// ---- Nodes/Algebraic Image Ops/Node_F_VN_BitwiseXorImagesExp.TcPOU
{attribute 'linkalways'} 
{attribute 'no_explicit_call' := 'This FB is a CLASS and must be accessed using methods or properties'}
{attribute 'enable_dynamic_creation'}
FUNCTION_BLOCK Node_F_VN_BitwiseXorImagesExp EXTENDS VisionNode
VAR
    ipSrcImage1 : _ITcVnImage;
    ipSrcImage2 : _ITcVnImage;
    ipDestImage : _ITcVnImage;
    ipMask : _ITcVnImage;
    hrPrev : _HRESULT(S_OK);
	hresult : _HRESULT(S_OK);
END_VAR

METHOD PUBLIC  Clone : I_Node
VAR
	pNode : POINTER TO Node_F_VN_BitwiseXorImagesExp;
END_VAR
pNode := __NEW(Node_F_VN_BitwiseXorImagesExp);
Clone := pNode^;
END_METHOD

METHOD FB_init : BOOL
VAR_INPUT
	bInitRetains : BOOL; // if TRUE, the retain variables are initialized (warm start / cold start)
	bInCopyCode : BOOL;  // if TRUE, the instance afterwards gets moved into the copy code (online change)
END_VAR
AddInput('ipSrcImage1', ipSrcImage1);
AddInput('ipSrcImage2', ipSrcImage2);
AddInput('ipMask', ipMask);
AddInput('hrPrev', hrPrev);
AddOutput('ipDestImage', ipDestImage);
AddOutput('hresult',hresult);
END_METHOD

METHOD PROTECTED OnExecute
hresult.Value := F_VN_BitwiseXorImagesExp(
    ipSrcImage1 := ipSrcImage1.Value,
    ipSrcImage2 := ipSrcImage2.Value,
	ipDestImage := ipDestImage.Value,
    ipMask := ipMask.Value,
	hrPrev:= hrPrev.Value);
END_METHOD

METHOD PUBLIC PreExecutionCheck
VAR_INPUT
	Check : I_PreExecutionChecks;
END_VAR
Check.IsTrue(ipSrcImage1.IsValid, 'ipSrcImage1 must contain an image');
Check.IsTrue(ipSrcImage2.IsValid, 'ipSrcImage2 must contain an image');
Check.IsTrue(IsImage1SizeEqualToImage2Size(ipSrcImage1.Value, ipSrcImage2.Value), 'ipSrcImage1 must be the same size as ipSrcImage2');
Check.IsTrue(ipMask.IsValid, 'ipMask must contain an image');
Check.IsTrue(ipMask.HasChannelCount(1), 'ipMask must have 1 channel');
Check.IsTrue(ipMask.IsPixelDepth(8), 'ipMask must have 8 bit pixel depth');
Check.IsTrue(IsImage1SizeEqualToImage2Size(ipMask.Value, ipSrcImage1.Value), 'ipMask must be the same size as ipSrcImage1');
END_METHOD

END_FUNCTION_BLOCK

// ---- Nodes/Algebraic Image Ops/Node_F_VN_BitwiseOrImagesExp.TcPOU
{attribute 'linkalways'} 
{attribute 'no_explicit_call' := 'This FB is a CLASS and must be accessed using methods or properties'}
{attribute 'enable_dynamic_creation'}
FUNCTION_BLOCK Node_F_VN_BitwiseOrImagesExp EXTENDS VisionNode
VAR
    ipSrcImage1 : _ITcVnImage;
    ipSrcImage2 : _ITcVnImage;
    ipDestImage : _ITcVnImage;
    ipMask : _ITcVnImage;
    hrPrev : _HRESULT(S_OK);
	hresult : _HRESULT(S_OK);
END_VAR

METHOD PUBLIC  Clone : I_Node
VAR
	pNode : POINTER TO Node_F_VN_BitwiseOrImagesExp;
END_VAR
pNode := __NEW(Node_F_VN_BitwiseOrImagesExp);
Clone := pNode^;
END_METHOD

METHOD FB_init : BOOL
VAR_INPUT
	bInitRetains : BOOL; // if TRUE, the retain variables are initialized (warm start / cold start)
	bInCopyCode : BOOL;  // if TRUE, the instance afterwards gets moved into the copy code (online change)
END_VAR
AddInput('ipSrcImage1', ipSrcImage1);
AddInput('ipSrcImage2', ipSrcImage2);
AddInput('ipMask', ipMask);
AddInput('hrPrev', hrPrev);
AddOutput('ipDestImage', ipDestImage);
AddOutput('hresult',hresult);
END_METHOD

METHOD PROTECTED OnExecute
hresult.Value := F_VN_BitwiseOrImagesExp(
    ipSrcImage1 := ipSrcImage1.Value,
    ipSrcImage2 := ipSrcImage2.Value,
	ipDestImage := ipDestImage.Value,
    ipMask := ipMask.Value,
	hrPrev:= hrPrev.Value);
END_METHOD

METHOD PUBLIC PreExecutionCheck
VAR_INPUT
	Check : I_PreExecutionChecks;
END_VAR
Check.IsTrue(ipSrcImage1.IsValid, 'ipSrcImage1 must contain an image');
Check.IsTrue(ipSrcImage2.IsValid, 'ipSrcImage2 must contain an image');
Check.IsTrue(IsImage1SizeEqualToImage2Size(ipSrcImage1.Value, ipSrcImage2.Value), 'ipSrcImage1 must be the same size as ipSrcImage2');
Check.IsTrue(ipMask.IsValid, 'ipMask must contain an image');
Check.IsTrue(ipMask.HasChannelCount(1), 'ipMask must have 1 channel');
Check.IsTrue(ipMask.IsPixelDepth(8), 'ipMask must have 8 bit pixel depth');
Check.IsTrue(IsImage1SizeEqualToImage2Size(ipMask.Value, ipSrcImage1.Value), 'ipMask must be the same size as ipSrcImage1');
END_METHOD

END_FUNCTION_BLOCK

// ---- Nodes/Algebraic Image Ops/Node_F_VN_BitwiseAndScalarWithImage.TcPOU
{attribute 'linkalways'} 
{attribute 'no_explicit_call' := 'This FB is a CLASS and must be accessed using methods or properties'}
{attribute 'enable_dynamic_creation'}
FUNCTION_BLOCK Node_F_VN_BitwiseAndScalarWithImage EXTENDS VisionNode
VAR
    fScalar : _LREAL(0.0);
    ipSrcImage : _ITcVnImage;
    ipDestImage : _ITcVnImage;
    hrPrev : _HRESULT(S_OK);
	hresult : _HRESULT(S_OK);
END_VAR

METHOD PUBLIC  Clone : I_Node
VAR
	pNode : POINTER TO Node_F_VN_BitwiseAndScalarWithImage;
END_VAR
pNode := __NEW(Node_F_VN_BitwiseAndScalarWithImage);
Clone := pNode^;
END_METHOD

METHOD FB_init : BOOL
VAR_INPUT
	bInitRetains : BOOL; // if TRUE, the retain variables are initialized (warm start / cold start)
	bInCopyCode : BOOL;  // if TRUE, the instance afterwards gets moved into the copy code (online change)
END_VAR
AddParameter('fScalar', fScalar);
AddInput('ipSrcImage', ipSrcImage);
AddInput('hrPrev', hrPrev);
AddOutput('ipDestImage', ipDestImage);
AddOutput('hresult',hresult);
END_METHOD

METHOD PROTECTED OnExecute
hresult.Value := F_VN_BitwiseAndScalarWithImage(
    fScalar := fScalar.Value,
    ipSrcImage := ipSrcImage.Value,
	ipDestImage := ipDestImage.Value,
	hrPrev:= hrPrev.Value);
END_METHOD

METHOD PUBLIC PreExecutionCheck
VAR_INPUT
	Check : I_PreExecutionChecks;
END_VAR
Check.IsTrue(ipSrcImage.IsValid, 'ipSrcImage must contain an image');
END_METHOD

END_FUNCTION_BLOCK

// ---- Nodes/Algebraic Image Ops/Node_F_VN_BitwiseXorVectorWithImage.TcPOU
{attribute 'linkalways'} 
{attribute 'no_explicit_call' := 'This FB is a CLASS and must be accessed using methods or properties'}
{attribute 'enable_dynamic_creation'}
FUNCTION_BLOCK Node_F_VN_BitwiseXorVectorWithImage EXTENDS VisionNode
VAR
    aVector : _TcVnVector4_LREAL;
    ipSrcImage : _ITcVnImage;
    ipDestImage : _ITcVnImage;
    hrPrev : _HRESULT(S_OK);
	hresult : _HRESULT(S_OK);
END_VAR

METHOD PUBLIC  Clone : I_Node
VAR
	pNode : POINTER TO Node_F_VN_BitwiseXorVectorWithImage;
END_VAR
pNode := __NEW(Node_F_VN_BitwiseXorVectorWithImage);
Clone := pNode^;
END_METHOD

METHOD FB_init : BOOL
VAR_INPUT
	bInitRetains : BOOL; // if TRUE, the retain variables are initialized (warm start / cold start)
	bInCopyCode : BOOL;  // if TRUE, the instance afterwards gets moved into the copy code (online change)
END_VAR
AddInput('aVector', aVector);
AddInput('ipSrcImage', ipSrcImage);
AddInput('hrPrev', hrPrev);
AddOutput('ipDestImage', ipDestImage);
AddOutput('hresult',hresult);
END_METHOD

METHOD PROTECTED OnExecute
hresult.Value := F_VN_BitwiseXorVectorWithImage(
    aVector := aVector.Value,
    ipSrcImage := ipSrcImage.Value,
	ipDestImage := ipDestImage.Value,
	hrPrev:= hrPrev.Value);
END_METHOD

METHOD PUBLIC PreExecutionCheck
VAR_INPUT
	Check : I_PreExecutionChecks;
END_VAR
Check.IsTrue(ipSrcImage.IsValid, 'ipSrcImage must contain an image');
END_METHOD

END_FUNCTION_BLOCK

// ---- Nodes/Algebraic Image Ops/Node_F_VN_BitwiseXorScalarWithImage.TcPOU
{attribute 'linkalways'} 
{attribute 'no_explicit_call' := 'This FB is a CLASS and must be accessed using methods or properties'}
{attribute 'enable_dynamic_creation'}
FUNCTION_BLOCK Node_F_VN_BitwiseXorScalarWithImage EXTENDS VisionNode
VAR
    fScalar : _LREAL(0.0);
    ipSrcImage : _ITcVnImage;
    ipDestImage : _ITcVnImage;
    hrPrev : _HRESULT(S_OK);
	hresult : _HRESULT(S_OK);
END_VAR

METHOD PUBLIC  Clone : I_Node
VAR
	pNode : POINTER TO Node_F_VN_BitwiseXorScalarWithImage;
END_VAR
pNode := __NEW(Node_F_VN_BitwiseXorScalarWithImage);
Clone := pNode^;
END_METHOD

METHOD FB_init : BOOL
VAR_INPUT
	bInitRetains : BOOL; // if TRUE, the retain variables are initialized (warm start / cold start)
	bInCopyCode : BOOL;  // if TRUE, the instance afterwards gets moved into the copy code (online change)
END_VAR
AddParameter('fScalar', fScalar);
AddInput('ipSrcImage', ipSrcImage);
AddInput('hrPrev', hrPrev);
AddOutput('ipDestImage', ipDestImage);
AddOutput('hresult',hresult);
END_METHOD

METHOD PROTECTED OnExecute
hresult.Value := F_VN_BitwiseXorScalarWithImage(
    fScalar := fScalar.Value,
    ipSrcImage := ipSrcImage.Value,
	ipDestImage := ipDestImage.Value,
	hrPrev:= hrPrev.Value);
END_METHOD

METHOD PUBLIC PreExecutionCheck
VAR_INPUT
	Check : I_PreExecutionChecks;
END_VAR
Check.IsTrue(ipSrcImage.IsValid, 'ipSrcImage must contain an image');
END_METHOD

END_FUNCTION_BLOCK

// ---- Nodes/Algebraic Image Ops/Node_F_VN_BitwiseOrVectorWithImage.TcPOU
{attribute 'linkalways'} 
{attribute 'no_explicit_call' := 'This FB is a CLASS and must be accessed using methods or properties'}
{attribute 'enable_dynamic_creation'}
FUNCTION_BLOCK Node_F_VN_BitwiseOrVectorWithImage EXTENDS VisionNode
VAR
    aVector : _TcVnVector4_LREAL;
    ipSrcImage : _ITcVnImage;
    ipDestImage : _ITcVnImage;
    hrPrev : _HRESULT(S_OK);
	hresult : _HRESULT(S_OK);
END_VAR

METHOD PUBLIC  Clone : I_Node
VAR
	pNode : POINTER TO Node_F_VN_BitwiseOrVectorWithImage;
END_VAR
pNode := __NEW(Node_F_VN_BitwiseOrVectorWithImage);
Clone := pNode^;
END_METHOD

METHOD FB_init : BOOL
VAR_INPUT
	bInitRetains : BOOL; // if TRUE, the retain variables are initialized (warm start / cold start)
	bInCopyCode : BOOL;  // if TRUE, the instance afterwards gets moved into the copy code (online change)
END_VAR
AddInput('aVector', aVector);
AddInput('ipSrcImage', ipSrcImage);
AddInput('hrPrev', hrPrev);
AddOutput('ipDestImage', ipDestImage);
AddOutput('hresult',hresult);
END_METHOD

METHOD PROTECTED OnExecute
hresult.Value := F_VN_BitwiseOrVectorWithImage(
    aVector := aVector.Value,
    ipSrcImage := ipSrcImage.Value,
	ipDestImage := ipDestImage.Value,
	hrPrev:= hrPrev.Value);
END_METHOD

METHOD PUBLIC PreExecutionCheck
VAR_INPUT
	Check : I_PreExecutionChecks;
END_VAR
Check.IsTrue(ipSrcImage.IsValid, 'ipSrcImage must contain an image');
END_METHOD

END_FUNCTION_BLOCK

// ---- Nodes/Algebraic Image Ops/Node_F_VN_BitwiseOrScalarWithImage.TcPOU
{attribute 'linkalways'} 
{attribute 'no_explicit_call' := 'This FB is a CLASS and must be accessed using methods or properties'}
{attribute 'enable_dynamic_creation'}
FUNCTION_BLOCK Node_F_VN_BitwiseOrScalarWithImage EXTENDS VisionNode
VAR
    fScalar : _LREAL(0.0);
    ipSrcImage : _ITcVnImage;
    ipDestImage : _ITcVnImage;
    hrPrev : _HRESULT(S_OK);
	hresult : _HRESULT(S_OK);
END_VAR

METHOD PUBLIC  Clone : I_Node
VAR
	pNode : POINTER TO Node_F_VN_BitwiseOrScalarWithImage;
END_VAR
pNode := __NEW(Node_F_VN_BitwiseOrScalarWithImage);
Clone := pNode^;
END_METHOD

METHOD FB_init : BOOL
VAR_INPUT
	bInitRetains : BOOL; // if TRUE, the retain variables are initialized (warm start / cold start)
	bInCopyCode : BOOL;  // if TRUE, the instance afterwards gets moved into the copy code (online change)
END_VAR
AddParameter('fScalar', fScalar);
AddInput('ipSrcImage', ipSrcImage);
AddInput('hrPrev', hrPrev);
AddOutput('ipDestImage', ipDestImage);
AddOutput('hresult',hresult);
END_METHOD

METHOD PROTECTED OnExecute
hresult.Value := F_VN_BitwiseOrScalarWithImage(
    fScalar := fScalar.Value,
    ipSrcImage := ipSrcImage.Value,
	ipDestImage := ipDestImage.Value,
	hrPrev:= hrPrev.Value);
END_METHOD

METHOD PUBLIC PreExecutionCheck
VAR_INPUT
	Check : I_PreExecutionChecks;
END_VAR
Check.IsTrue(ipSrcImage.IsValid, 'ipSrcImage must contain an image');
END_METHOD

END_FUNCTION_BLOCK

// ---- Nodes/Algebraic Image Ops/Node_F_VN_BitwiseAndVectorWithImage.TcPOU
{attribute 'linkalways'} 
{attribute 'no_explicit_call' := 'This FB is a CLASS and must be accessed using methods or properties'}
{attribute 'enable_dynamic_creation'}
FUNCTION_BLOCK Node_F_VN_BitwiseAndVectorWithImage EXTENDS VisionNode
VAR
    aVector : _TcVnVector4_LREAL;
    ipSrcImage : _ITcVnImage;
    ipDestImage : _ITcVnImage;
    hrPrev : _HRESULT(S_OK);
	hresult : _HRESULT(S_OK);
END_VAR

METHOD PUBLIC  Clone : I_Node
VAR
	pNode : POINTER TO Node_F_VN_BitwiseAndVectorWithImage;
END_VAR
pNode := __NEW(Node_F_VN_BitwiseAndVectorWithImage);
Clone := pNode^;
END_METHOD

METHOD FB_init : BOOL
VAR_INPUT
	bInitRetains : BOOL; // if TRUE, the retain variables are initialized (warm start / cold start)
	bInCopyCode : BOOL;  // if TRUE, the instance afterwards gets moved into the copy code (online change)
END_VAR
AddInput('aVector', aVector);
AddInput('ipSrcImage', ipSrcImage);
AddInput('hrPrev', hrPrev);
AddOutput('ipDestImage', ipDestImage);
AddOutput('hresult',hresult);
END_METHOD

METHOD PROTECTED OnExecute
hresult.Value := F_VN_BitwiseAndVectorWithImage(
    aVector := aVector.Value,
    ipSrcImage := ipSrcImage.Value,
	ipDestImage := ipDestImage.Value,
	hrPrev:= hrPrev.Value);
END_METHOD

METHOD PUBLIC PreExecutionCheck
VAR_INPUT
	Check : I_PreExecutionChecks;
END_VAR
Check.IsTrue(ipSrcImage.IsValid, 'ipSrcImage must contain an image');
END_METHOD

END_FUNCTION_BLOCK

// ---- Nodes/Algebraic Image Ops/Node_F_VN_DivideImageByScalar.TcPOU
{attribute 'linkalways'} 
{attribute 'no_explicit_call' := 'This FB is a CLASS and must be accessed using methods or properties'}
{attribute 'enable_dynamic_creation'}
FUNCTION_BLOCK Node_F_VN_DivideImageByScalar EXTENDS VisionNode
VAR
    ipSrcImage : _ITcVnImage;
    fScalar : _LREAL(0.0);
    ipDestImage : _ITcVnImage;
    hrPrev : _HRESULT(S_OK);
	hresult : _HRESULT(S_OK);
END_VAR

METHOD PUBLIC  Clone : I_Node
VAR
	pNode : POINTER TO Node_F_VN_DivideImageByScalar;
END_VAR
pNode := __NEW(Node_F_VN_DivideImageByScalar);
Clone := pNode^;
END_METHOD

METHOD FB_init : BOOL
VAR_INPUT
	bInitRetains : BOOL; // if TRUE, the retain variables are initialized (warm start / cold start)
	bInCopyCode : BOOL;  // if TRUE, the instance afterwards gets moved into the copy code (online change)
END_VAR
AddInput('ipSrcImage', ipSrcImage);
AddParameter('fScalar', fScalar);
AddInput('hrPrev', hrPrev);
AddOutput('ipDestImage', ipDestImage);
AddOutput('hresult',hresult);
END_METHOD

METHOD PROTECTED OnExecute
hresult.Value := F_VN_DivideImageByScalar(
    ipSrcImage := ipSrcImage.Value,
    fScalar := fScalar.Value,
	ipDestImage := ipDestImage.Value,
	hrPrev:= hrPrev.Value);
END_METHOD

METHOD PUBLIC PreExecutionCheck
VAR_INPUT
	Check : I_PreExecutionChecks;
END_VAR
Check.IsTrue(ipSrcImage.IsValid, 'ipSrcImage must contain an image');
END_METHOD

END_FUNCTION_BLOCK

// ---- Nodes/Algebraic Image Ops/Node_F_VN_DivideVectorByImage.TcPOU
{attribute 'linkalways'} 
{attribute 'no_explicit_call' := 'This FB is a CLASS and must be accessed using methods or properties'}
{attribute 'enable_dynamic_creation'}
FUNCTION_BLOCK Node_F_VN_DivideVectorByImage EXTENDS VisionNode
VAR
    aVector : _TcVnVector4_LREAL;
    ipSrcImage : _ITcVnImage;
    ipDestImage : _ITcVnImage;
    hrPrev : _HRESULT(S_OK);
	hresult : _HRESULT(S_OK);
END_VAR

METHOD PUBLIC  Clone : I_Node
VAR
	pNode : POINTER TO Node_F_VN_DivideVectorByImage;
END_VAR
pNode := __NEW(Node_F_VN_DivideVectorByImage);
Clone := pNode^;
END_METHOD

METHOD FB_init : BOOL
VAR_INPUT
	bInitRetains : BOOL; // if TRUE, the retain variables are initialized (warm start / cold start)
	bInCopyCode : BOOL;  // if TRUE, the instance afterwards gets moved into the copy code (online change)
END_VAR
AddInput('aVector', aVector);
AddInput('ipSrcImage', ipSrcImage);
AddInput('hrPrev', hrPrev);
AddOutput('ipDestImage', ipDestImage);
AddOutput('hresult',hresult);
END_METHOD

METHOD PROTECTED OnExecute
hresult.Value := F_VN_DivideVectorByImage(
    aVector := aVector.Value,
    ipSrcImage := ipSrcImage.Value,
	ipDestImage := ipDestImage.Value,
	hrPrev:= hrPrev.Value);
END_METHOD

METHOD PUBLIC PreExecutionCheck
VAR_INPUT
	Check : I_PreExecutionChecks;
END_VAR
Check.IsTrue(ipSrcImage.IsValid, 'ipSrcImage must contain an image');
END_METHOD

END_FUNCTION_BLOCK

// ---- Nodes/Algebraic Image Ops/Node_F_VN_DivideScalarByImage.TcPOU
{attribute 'linkalways'} 
{attribute 'no_explicit_call' := 'This FB is a CLASS and must be accessed using methods or properties'}
{attribute 'enable_dynamic_creation'}
FUNCTION_BLOCK Node_F_VN_DivideScalarByImage EXTENDS VisionNode
VAR
    fScalar : _LREAL(0.0);
    ipSrcImage : _ITcVnImage;
    ipDestImage : _ITcVnImage;
    hrPrev : _HRESULT(S_OK);
	hresult : _HRESULT(S_OK);
END_VAR

METHOD PUBLIC  Clone : I_Node
VAR
	pNode : POINTER TO Node_F_VN_DivideScalarByImage;
END_VAR
pNode := __NEW(Node_F_VN_DivideScalarByImage);
Clone := pNode^;
END_METHOD

METHOD FB_init : BOOL
VAR_INPUT
	bInitRetains : BOOL; // if TRUE, the retain variables are initialized (warm start / cold start)
	bInCopyCode : BOOL;  // if TRUE, the instance afterwards gets moved into the copy code (online change)
END_VAR
AddParameter('fScalar', fScalar);
AddInput('ipSrcImage', ipSrcImage);
AddInput('hrPrev', hrPrev);
AddOutput('ipDestImage', ipDestImage);
AddOutput('hresult',hresult);
END_METHOD

METHOD PROTECTED OnExecute
hresult.Value := F_VN_DivideScalarByImage(
    fScalar := fScalar.Value,
    ipSrcImage := ipSrcImage.Value,
	ipDestImage := ipDestImage.Value,
	hrPrev:= hrPrev.Value);
END_METHOD

METHOD PUBLIC PreExecutionCheck
VAR_INPUT
	Check : I_PreExecutionChecks;
END_VAR
Check.IsTrue(ipSrcImage.IsValid, 'ipSrcImage must contain an image');
END_METHOD

END_FUNCTION_BLOCK

// ---- Nodes/Algebraic Image Ops/Node_F_VN_DivideImageByVector.TcPOU
{attribute 'linkalways'} 
{attribute 'no_explicit_call' := 'This FB is a CLASS and must be accessed using methods or properties'}
{attribute 'enable_dynamic_creation'}
FUNCTION_BLOCK Node_F_VN_DivideImageByVector EXTENDS VisionNode
VAR
    ipSrcImage : _ITcVnImage;
    aVector : _TcVnVector4_LREAL;
    ipDestImage : _ITcVnImage;
    hrPrev : _HRESULT(S_OK);
	hresult : _HRESULT(S_OK);
END_VAR

METHOD PUBLIC  Clone : I_Node
VAR
	pNode : POINTER TO Node_F_VN_DivideImageByVector;
END_VAR
pNode := __NEW(Node_F_VN_DivideImageByVector);
Clone := pNode^;
END_METHOD

METHOD FB_init : BOOL
VAR_INPUT
	bInitRetains : BOOL; // if TRUE, the retain variables are initialized (warm start / cold start)
	bInCopyCode : BOOL;  // if TRUE, the instance afterwards gets moved into the copy code (online change)
END_VAR
AddInput('ipSrcImage', ipSrcImage);
AddInput('aVector', aVector);
AddInput('hrPrev', hrPrev);
AddOutput('ipDestImage', ipDestImage);
AddOutput('hresult',hresult);
END_METHOD

METHOD PROTECTED OnExecute
hresult.Value := F_VN_DivideImageByVector(
    ipSrcImage := ipSrcImage.Value,
    aVector := aVector.Value,
	ipDestImage := ipDestImage.Value,
	hrPrev:= hrPrev.Value);
END_METHOD

METHOD PUBLIC PreExecutionCheck
VAR_INPUT
	Check : I_PreExecutionChecks;
END_VAR
Check.IsTrue(ipSrcImage.IsValid, 'ipSrcImage must contain an image');
END_METHOD

END_FUNCTION_BLOCK

// ---- Nodes/Algebraic Image Ops/Node_F_VN_ElementwiseExp.TcPOU
{attribute 'linkalways'} 
{attribute 'no_explicit_call' := 'This FB is a CLASS and must be accessed using methods or properties'}
{attribute 'enable_dynamic_creation'}
FUNCTION_BLOCK Node_F_VN_ElementwiseExp EXTENDS VisionNode
VAR
    ipSrcImage : _ITcVnImage;
    ipDestImage : _ITcVnImage;
    hrPrev : _HRESULT(S_OK);
	hresult : _HRESULT(S_OK);
END_VAR

METHOD PUBLIC  Clone : I_Node
VAR
	pNode : POINTER TO Node_F_VN_ElementwiseExp;
END_VAR
pNode := __NEW(Node_F_VN_ElementwiseExp);
Clone := pNode^;
END_METHOD

METHOD FB_init : BOOL
VAR_INPUT
	bInitRetains : BOOL; // if TRUE, the retain variables are initialized (warm start / cold start)
	bInCopyCode : BOOL;  // if TRUE, the instance afterwards gets moved into the copy code (online change)
END_VAR
AddInput('ipSrcImage', ipSrcImage);
AddInput('hrPrev', hrPrev);
AddOutput('ipDestImage', ipDestImage);
AddOutput('hresult',hresult);
END_METHOD

METHOD PROTECTED OnExecute
hresult.Value := F_VN_ElementwiseExp(
    ipSrcImage := ipSrcImage.Value,
	ipDestImage := ipDestImage.Value,
	hrPrev:= hrPrev.Value);
END_METHOD

METHOD PUBLIC PreExecutionCheck
VAR_INPUT
	Check : I_PreExecutionChecks;
END_VAR
Check.IsTrue(ipSrcImage.IsValid, 'ipSrcImage must contain an image');
Check.IsTrue((ipSrcImage.IsPixelDepth(32) OR
              ipSrcImage.IsPixelDepth(64)), 'ipSrcImage must have 32 or 64 bit pixel depth');
END_METHOD

END_FUNCTION_BLOCK

// ---- Nodes/Algebraic Image Ops/Node_F_VN_ElementwiseLog.TcPOU
{attribute 'linkalways'} 
{attribute 'no_explicit_call' := 'This FB is a CLASS and must be accessed using methods or properties'}
{attribute 'enable_dynamic_creation'}
FUNCTION_BLOCK Node_F_VN_ElementwiseLog EXTENDS VisionNode
VAR
    ipSrcImage : _ITcVnImage;
    ipDestImage : _ITcVnImage;
    hrPrev : _HRESULT(S_OK);
	hresult : _HRESULT(S_OK);
END_VAR

METHOD PUBLIC  Clone : I_Node
VAR
	pNode : POINTER TO Node_F_VN_ElementwiseLog;
END_VAR
pNode := __NEW(Node_F_VN_ElementwiseLog);
Clone := pNode^;
END_METHOD

METHOD FB_init : BOOL
VAR_INPUT
	bInitRetains : BOOL; // if TRUE, the retain variables are initialized (warm start / cold start)
	bInCopyCode : BOOL;  // if TRUE, the instance afterwards gets moved into the copy code (online change)
END_VAR
AddInput('ipSrcImage', ipSrcImage);
AddInput('hrPrev', hrPrev);
AddOutput('ipDestImage', ipDestImage);
AddOutput('hresult',hresult);
END_METHOD

METHOD PROTECTED OnExecute
hresult.Value := F_VN_ElementwiseLog(
    ipSrcImage := ipSrcImage.Value,
	ipDestImage := ipDestImage.Value,
	hrPrev:= hrPrev.Value);
END_METHOD

METHOD PUBLIC PreExecutionCheck
VAR_INPUT
	Check : I_PreExecutionChecks;
END_VAR
Check.IsTrue(ipSrcImage.IsValid, 'ipSrcImage must contain an image');
Check.IsTrue((ipSrcImage.IsPixelDepth(32) OR
              ipSrcImage.IsPixelDepth(64)), 'ipSrcImage must have 32 or 64 bit pixel depth');
END_METHOD

END_FUNCTION_BLOCK

// ---- Nodes/Algebraic Image Ops/Node_F_VN_MaxImageWithScalarExp.TcPOU
{attribute 'linkalways'} 
{attribute 'no_explicit_call' := 'This FB is a CLASS and must be accessed using methods or properties'}
{attribute 'enable_dynamic_creation'}
FUNCTION_BLOCK Node_F_VN_MaxImageWithScalarExp EXTENDS VisionNode
VAR
    fScalar : _LREAL(0.0);
    ipSrcImage : _ITcVnImage;
    ipDestImage : _ITcVnImage;
    ipMask : _ITcVnImage;
    hrPrev : _HRESULT(S_OK);
	hresult : _HRESULT(S_OK);
END_VAR

METHOD PUBLIC  Clone : I_Node
VAR
	pNode : POINTER TO Node_F_VN_MaxImageWithScalarExp;
END_VAR
pNode := __NEW(Node_F_VN_MaxImageWithScalarExp);
Clone := pNode^;
END_METHOD

METHOD FB_init : BOOL
VAR_INPUT
	bInitRetains : BOOL; // if TRUE, the retain variables are initialized (warm start / cold start)
	bInCopyCode : BOOL;  // if TRUE, the instance afterwards gets moved into the copy code (online change)
END_VAR
AddParameter('fScalar', fScalar);
AddInput('ipSrcImage', ipSrcImage);
AddInput('ipMask', ipMask);
AddInput('hrPrev', hrPrev);
AddOutput('ipDestImage', ipDestImage);
AddOutput('hresult',hresult);
END_METHOD

METHOD PROTECTED OnExecute
hresult.Value := F_VN_MaxImageWithScalarExp(
    fScalar := fScalar.Value,
    ipSrcImage := ipSrcImage.Value,
	ipDestImage := ipDestImage.Value,
    ipMask := ipMask.Value,
	hrPrev:= hrPrev.Value);
END_METHOD

METHOD PUBLIC PreExecutionCheck
VAR_INPUT
	Check : I_PreExecutionChecks;
END_VAR
Check.IsTrue(ipSrcImage.IsValid, 'ipSrcImage must contain an image');
Check.IsTrue(ipMask.IsValid, 'ipMask must contain an image');
Check.IsTrue(ipMask.HasChannelCount(1), 'ipMask must have 1 channel');
Check.IsTrue(ipMask.IsPixelDepth(8), 'ipMask must have 8 bit pixel depth');
Check.IsTrue(IsImage1SizeEqualToImage2Size(ipMask.Value, ipSrcImage.Value), 'ipMask must be the same size as ipSrcImage');
END_METHOD

END_FUNCTION_BLOCK

// ---- Nodes/Algebraic Image Ops/Node_F_VN_MaxImageWithVectorExp.TcPOU
{attribute 'linkalways'} 
{attribute 'no_explicit_call' := 'This FB is a CLASS and must be accessed using methods or properties'}
{attribute 'enable_dynamic_creation'}
FUNCTION_BLOCK Node_F_VN_MaxImageWithVectorExp EXTENDS VisionNode
VAR
    aVector : _TcVnVector4_LREAL;
    ipSrcImage : _ITcVnImage;
    ipDestImage : _ITcVnImage;
    ipMask : _ITcVnImage;
    hrPrev : _HRESULT(S_OK);
	hresult : _HRESULT(S_OK);
END_VAR

METHOD PUBLIC  Clone : I_Node
VAR
	pNode : POINTER TO Node_F_VN_MaxImageWithVectorExp;
END_VAR
pNode := __NEW(Node_F_VN_MaxImageWithVectorExp);
Clone := pNode^;
END_METHOD

METHOD FB_init : BOOL
VAR_INPUT
	bInitRetains : BOOL; // if TRUE, the retain variables are initialized (warm start / cold start)
	bInCopyCode : BOOL;  // if TRUE, the instance afterwards gets moved into the copy code (online change)
END_VAR
AddInput('aVector', aVector);
AddInput('ipSrcImage', ipSrcImage);
AddInput('ipMask', ipMask);
AddInput('hrPrev', hrPrev);
AddOutput('ipDestImage', ipDestImage);
AddOutput('hresult',hresult);
END_METHOD

METHOD PROTECTED OnExecute
hresult.Value := F_VN_MaxImageWithVectorExp(
    aVector := aVector.Value,
    ipSrcImage := ipSrcImage.Value,
	ipDestImage := ipDestImage.Value,
    ipMask := ipMask.Value,
	hrPrev:= hrPrev.Value);
END_METHOD

METHOD PUBLIC PreExecutionCheck
VAR_INPUT
	Check : I_PreExecutionChecks;
END_VAR
Check.IsTrue(ipSrcImage.IsValid, 'ipSrcImage must contain an image');
Check.IsTrue(ipMask.IsValid, 'ipMask must contain an image');
Check.IsTrue(ipMask.HasChannelCount(1), 'ipMask must have 1 channel');
Check.IsTrue(ipMask.IsPixelDepth(8), 'ipMask must have 8 bit pixel depth');
Check.IsTrue(IsImage1SizeEqualToImage2Size(ipMask.Value, ipSrcImage.Value), 'ipMask must be the same size as ipSrcImage');
END_METHOD

END_FUNCTION_BLOCK

// ---- Nodes/Algebraic Image Ops/Node_F_VN_MinImageWithVectorExp.TcPOU
{attribute 'linkalways'} 
{attribute 'no_explicit_call' := 'This FB is a CLASS and must be accessed using methods or properties'}
{attribute 'enable_dynamic_creation'}
FUNCTION_BLOCK Node_F_VN_MinImageWithVectorExp EXTENDS VisionNode
VAR
    aVector : _TcVnVector4_LREAL;
    ipSrcImage : _ITcVnImage;
    ipDestImage : _ITcVnImage;
    ipMask : _ITcVnImage;
    hrPrev : _HRESULT(S_OK);
	hresult : _HRESULT(S_OK);
END_VAR

METHOD PUBLIC  Clone : I_Node
VAR
	pNode : POINTER TO Node_F_VN_MinImageWithVectorExp;
END_VAR
pNode := __NEW(Node_F_VN_MinImageWithVectorExp);
Clone := pNode^;
END_METHOD

METHOD FB_init : BOOL
VAR_INPUT
	bInitRetains : BOOL; // if TRUE, the retain variables are initialized (warm start / cold start)
	bInCopyCode : BOOL;  // if TRUE, the instance afterwards gets moved into the copy code (online change)
END_VAR
AddInput('aVector', aVector);
AddInput('ipSrcImage', ipSrcImage);
AddInput('ipMask', ipMask);
AddInput('hrPrev', hrPrev);
AddOutput('ipDestImage', ipDestImage);
AddOutput('hresult',hresult);
END_METHOD

METHOD PROTECTED OnExecute
hresult.Value := F_VN_MinImageWithVectorExp(
    aVector := aVector.Value,
    ipSrcImage := ipSrcImage.Value,
	ipDestImage := ipDestImage.Value,
    ipMask := ipMask.Value,
	hrPrev:= hrPrev.Value);
END_METHOD

METHOD PUBLIC PreExecutionCheck
VAR_INPUT
	Check : I_PreExecutionChecks;
END_VAR
Check.IsTrue(ipSrcImage.IsValid, 'ipSrcImage must contain an image');
Check.IsTrue(ipMask.IsValid, 'ipMask must contain an image');
Check.IsTrue(ipMask.HasChannelCount(1), 'ipMask must have 1 channel');
Check.IsTrue(ipMask.IsPixelDepth(8), 'ipMask must have 8 bit pixel depth');
Check.IsTrue(IsImage1SizeEqualToImage2Size(ipMask.Value, ipSrcImage.Value), 'ipMask must be the same size as ipSrcImage');
END_METHOD

END_FUNCTION_BLOCK

// ---- Nodes/Algebraic Image Ops/Node_F_VN_MinImageWithScalarExp.TcPOU
{attribute 'linkalways'} 
{attribute 'no_explicit_call' := 'This FB is a CLASS and must be accessed using methods or properties'}
{attribute 'enable_dynamic_creation'}
FUNCTION_BLOCK Node_F_VN_MinImageWithScalarExp EXTENDS VisionNode
VAR
    fScalar : _LREAL(0.0);
    ipSrcImage : _ITcVnImage;
    ipDestImage : _ITcVnImage;
    ipMask : _ITcVnImage;
    hrPrev : _HRESULT(S_OK);
	hresult : _HRESULT(S_OK);
END_VAR

METHOD PUBLIC  Clone : I_Node
VAR
	pNode : POINTER TO Node_F_VN_MinImageWithScalarExp;
END_VAR
pNode := __NEW(Node_F_VN_MinImageWithScalarExp);
Clone := pNode^;
END_METHOD

METHOD FB_init : BOOL
VAR_INPUT
	bInitRetains : BOOL; // if TRUE, the retain variables are initialized (warm start / cold start)
	bInCopyCode : BOOL;  // if TRUE, the instance afterwards gets moved into the copy code (online change)
END_VAR
AddParameter('fScalar', fScalar);
AddInput('ipSrcImage', ipSrcImage);
AddInput('ipMask', ipMask);
AddInput('hrPrev', hrPrev);
AddOutput('ipDestImage', ipDestImage);
AddOutput('hresult',hresult);
END_METHOD

METHOD PROTECTED OnExecute
hresult.Value := F_VN_MinImageWithScalarExp(
    fScalar := fScalar.Value,
    ipSrcImage := ipSrcImage.Value,
	ipDestImage := ipDestImage.Value,
    ipMask := ipMask.Value,
	hrPrev:= hrPrev.Value);
END_METHOD

METHOD PUBLIC PreExecutionCheck
VAR_INPUT
	Check : I_PreExecutionChecks;
END_VAR
Check.IsTrue(ipSrcImage.IsValid, 'ipSrcImage must contain an image');
Check.IsTrue(ipMask.IsValid, 'ipMask must contain an image');
Check.IsTrue(ipMask.HasChannelCount(1), 'ipMask must have 1 channel');
Check.IsTrue(ipMask.IsPixelDepth(8), 'ipMask must have 8 bit pixel depth');
Check.IsTrue(IsImage1SizeEqualToImage2Size(ipMask.Value, ipSrcImage.Value), 'ipMask must be the same size as ipSrcImage');
END_METHOD

END_FUNCTION_BLOCK

// ---- Nodes/Algebraic Image Ops/Node_F_VN_MinImageExp.TcPOU
{attribute 'linkalways'} 
{attribute 'no_explicit_call' := 'This FB is a CLASS and must be accessed using methods or properties'}
{attribute 'enable_dynamic_creation'}
FUNCTION_BLOCK Node_F_VN_MinImageExp EXTENDS VisionNode
VAR
    ipSrcImage1 : _ITcVnImage;
    ipSrcImage2 : _ITcVnImage;
    ipDestImage : _ITcVnImage;
    ipMask : _ITcVnImage;
    hrPrev : _HRESULT(S_OK);
	hresult : _HRESULT(S_OK);
END_VAR

METHOD PUBLIC  Clone : I_Node
VAR
	pNode : POINTER TO Node_F_VN_MinImageExp;
END_VAR
pNode := __NEW(Node_F_VN_MinImageExp);
Clone := pNode^;
END_METHOD

METHOD FB_init : BOOL
VAR_INPUT
	bInitRetains : BOOL; // if TRUE, the retain variables are initialized (warm start / cold start)
	bInCopyCode : BOOL;  // if TRUE, the instance afterwards gets moved into the copy code (online change)
END_VAR
AddInput('ipSrcImage1', ipSrcImage1);
AddInput('ipSrcImage2', ipSrcImage2);
AddInput('ipMask', ipMask);
AddInput('hrPrev', hrPrev);
AddOutput('ipDestImage', ipDestImage);
AddOutput('hresult',hresult);
END_METHOD

METHOD PROTECTED OnExecute
hresult.Value := F_VN_MinImageExp(
    ipSrcImage1 := ipSrcImage1.Value,
    ipSrcImage2 := ipSrcImage2.Value,
	ipDestImage := ipDestImage.Value,
    ipMask := ipMask.Value,
	hrPrev:= hrPrev.Value);
END_METHOD

METHOD PUBLIC PreExecutionCheck
VAR_INPUT
	Check : I_PreExecutionChecks;
END_VAR
Check.IsTrue(ipSrcImage1.IsValid, 'ipSrcImage1 must contain an image');
Check.IsTrue(ipSrcImage2.IsValid, 'ipSrcImage2 must contain an image');
Check.IsTrue(IsImage1SizeEqualToImage2Size(ipSrcImage1.Value, ipSrcImage2.Value), 'ipSrcImage1 must be the same size as ipSrcImage2');
Check.IsTrue(ipMask.IsValid, 'ipMask must contain an image');
Check.IsTrue(ipMask.HasChannelCount(1), 'ipMask must have 1 channel');
Check.IsTrue(ipMask.IsPixelDepth(8), 'ipMask must have 8 bit pixel depth');
Check.IsTrue(IsImage1SizeEqualToImage2Size(ipMask.Value, ipSrcImage1.Value), 'ipMask must be the same size as ipSrcImage1');
END_METHOD

END_FUNCTION_BLOCK

// ---- Nodes/Algebraic Image Ops/Node_F_VN_MaxImageWithScalar.TcPOU
{attribute 'linkalways'} 
{attribute 'no_explicit_call' := 'This FB is a CLASS and must be accessed using methods or properties'}
{attribute 'enable_dynamic_creation'}
FUNCTION_BLOCK Node_F_VN_MaxImageWithScalar EXTENDS VisionNode
VAR
    fScalar : _LREAL(0.0);
    ipSrcImage : _ITcVnImage;
    ipDestImage : _ITcVnImage;
    hrPrev : _HRESULT(S_OK);
	hresult : _HRESULT(S_OK);
END_VAR

METHOD PUBLIC  Clone : I_Node
VAR
	pNode : POINTER TO Node_F_VN_MaxImageWithScalar;
END_VAR
pNode := __NEW(Node_F_VN_MaxImageWithScalar);
Clone := pNode^;
END_METHOD

METHOD FB_init : BOOL
VAR_INPUT
	bInitRetains : BOOL; // if TRUE, the retain variables are initialized (warm start / cold start)
	bInCopyCode : BOOL;  // if TRUE, the instance afterwards gets moved into the copy code (online change)
END_VAR
AddParameter('fScalar', fScalar);
AddInput('ipSrcImage', ipSrcImage);
AddInput('hrPrev', hrPrev);
AddOutput('ipDestImage', ipDestImage);
AddOutput('hresult',hresult);
END_METHOD

METHOD PROTECTED OnExecute
hresult.Value := F_VN_MaxImageWithScalar(
    fScalar := fScalar.Value,
    ipSrcImage := ipSrcImage.Value,
	ipDestImage := ipDestImage.Value,
	hrPrev:= hrPrev.Value);
END_METHOD

METHOD PUBLIC PreExecutionCheck
VAR_INPUT
	Check : I_PreExecutionChecks;
END_VAR
Check.IsTrue(ipSrcImage.IsValid, 'ipSrcImage must contain an image');
END_METHOD

END_FUNCTION_BLOCK

// ---- Nodes/Algebraic Image Ops/Node_F_VN_MinImageWithVector.TcPOU
{attribute 'linkalways'} 
{attribute 'no_explicit_call' := 'This FB is a CLASS and must be accessed using methods or properties'}
{attribute 'enable_dynamic_creation'}
FUNCTION_BLOCK Node_F_VN_MinImageWithVector EXTENDS VisionNode
VAR
    aVector : _TcVnVector4_LREAL;
    ipSrcImage : _ITcVnImage;
    ipDestImage : _ITcVnImage;
    hrPrev : _HRESULT(S_OK);
	hresult : _HRESULT(S_OK);
END_VAR

METHOD PUBLIC  Clone : I_Node
VAR
	pNode : POINTER TO Node_F_VN_MinImageWithVector;
END_VAR
pNode := __NEW(Node_F_VN_MinImageWithVector);
Clone := pNode^;
END_METHOD

METHOD FB_init : BOOL
VAR_INPUT
	bInitRetains : BOOL; // if TRUE, the retain variables are initialized (warm start / cold start)
	bInCopyCode : BOOL;  // if TRUE, the instance afterwards gets moved into the copy code (online change)
END_VAR
AddInput('aVector', aVector);
AddInput('ipSrcImage', ipSrcImage);
AddInput('hrPrev', hrPrev);
AddOutput('ipDestImage', ipDestImage);
AddOutput('hresult',hresult);
END_METHOD

METHOD PROTECTED OnExecute
hresult.Value := F_VN_MinImageWithVector(
    aVector := aVector.Value,
    ipSrcImage := ipSrcImage.Value,
	ipDestImage := ipDestImage.Value,
	hrPrev:= hrPrev.Value);
END_METHOD

METHOD PUBLIC PreExecutionCheck
VAR_INPUT
	Check : I_PreExecutionChecks;
END_VAR
Check.IsTrue(ipSrcImage.IsValid, 'ipSrcImage must contain an image');
END_METHOD

END_FUNCTION_BLOCK

// ---- Nodes/Algebraic Image Ops/Node_F_VN_MinImageWithScalar.TcPOU
{attribute 'linkalways'} 
{attribute 'no_explicit_call' := 'This FB is a CLASS and must be accessed using methods or properties'}
{attribute 'enable_dynamic_creation'}
FUNCTION_BLOCK Node_F_VN_MinImageWithScalar EXTENDS VisionNode
VAR
    fScalar : _LREAL(0.0);
    ipSrcImage : _ITcVnImage;
    ipDestImage : _ITcVnImage;
    hrPrev : _HRESULT(S_OK);
	hresult : _HRESULT(S_OK);
END_VAR

METHOD PUBLIC  Clone : I_Node
VAR
	pNode : POINTER TO Node_F_VN_MinImageWithScalar;
END_VAR
pNode := __NEW(Node_F_VN_MinImageWithScalar);
Clone := pNode^;
END_METHOD

METHOD FB_init : BOOL
VAR_INPUT
	bInitRetains : BOOL; // if TRUE, the retain variables are initialized (warm start / cold start)
	bInCopyCode : BOOL;  // if TRUE, the instance afterwards gets moved into the copy code (online change)
END_VAR
AddParameter('fScalar', fScalar);
AddInput('ipSrcImage', ipSrcImage);
AddInput('hrPrev', hrPrev);
AddOutput('ipDestImage', ipDestImage);
AddOutput('hresult',hresult);
END_METHOD

METHOD PROTECTED OnExecute
hresult.Value := F_VN_MinImageWithScalar(
    fScalar := fScalar.Value,
    ipSrcImage := ipSrcImage.Value,
	ipDestImage := ipDestImage.Value,
	hrPrev:= hrPrev.Value);
END_METHOD

METHOD PUBLIC PreExecutionCheck
VAR_INPUT
	Check : I_PreExecutionChecks;
END_VAR
Check.IsTrue(ipSrcImage.IsValid, 'ipSrcImage must contain an image');
END_METHOD

END_FUNCTION_BLOCK

// ---- Nodes/Algebraic Image Ops/Node_F_VN_MaxImageWithVector.TcPOU
{attribute 'linkalways'} 
{attribute 'no_explicit_call' := 'This FB is a CLASS and must be accessed using methods or properties'}
{attribute 'enable_dynamic_creation'}
FUNCTION_BLOCK Node_F_VN_MaxImageWithVector EXTENDS VisionNode
VAR
    aVector : _TcVnVector4_LREAL;
    ipSrcImage : _ITcVnImage;
    ipDestImage : _ITcVnImage;
    hrPrev : _HRESULT(S_OK);
	hresult : _HRESULT(S_OK);
END_VAR

METHOD PUBLIC  Clone : I_Node
VAR
	pNode : POINTER TO Node_F_VN_MaxImageWithVector;
END_VAR
pNode := __NEW(Node_F_VN_MaxImageWithVector);
Clone := pNode^;
END_METHOD

METHOD FB_init : BOOL
VAR_INPUT
	bInitRetains : BOOL; // if TRUE, the retain variables are initialized (warm start / cold start)
	bInCopyCode : BOOL;  // if TRUE, the instance afterwards gets moved into the copy code (online change)
END_VAR
AddInput('aVector', aVector);
AddInput('ipSrcImage', ipSrcImage);
AddInput('hrPrev', hrPrev);
AddOutput('ipDestImage', ipDestImage);
AddOutput('hresult',hresult);
END_METHOD

METHOD PROTECTED OnExecute
hresult.Value := F_VN_MaxImageWithVector(
    aVector := aVector.Value,
    ipSrcImage := ipSrcImage.Value,
	ipDestImage := ipDestImage.Value,
	hrPrev:= hrPrev.Value);
END_METHOD

METHOD PUBLIC PreExecutionCheck
VAR_INPUT
	Check : I_PreExecutionChecks;
END_VAR
Check.IsTrue(ipSrcImage.IsValid, 'ipSrcImage must contain an image');
END_METHOD

END_FUNCTION_BLOCK

// ---- Nodes/Algebraic Image Ops/Node_F_VN_MultiplyImageWithScalar.TcPOU
{attribute 'linkalways'} 
{attribute 'no_explicit_call' := 'This FB is a CLASS and must be accessed using methods or properties'}
{attribute 'enable_dynamic_creation'}
FUNCTION_BLOCK Node_F_VN_MultiplyImageWithScalar EXTENDS VisionNode
VAR
    fScalar : _LREAL(0.0);
    ipSrcImage : _ITcVnImage;
    ipDestImage : _ITcVnImage;
    hrPrev : _HRESULT(S_OK);
	hresult : _HRESULT(S_OK);
END_VAR

METHOD PUBLIC  Clone : I_Node
VAR
	pNode : POINTER TO Node_F_VN_MultiplyImageWithScalar;
END_VAR
pNode := __NEW(Node_F_VN_MultiplyImageWithScalar);
Clone := pNode^;
END_METHOD

METHOD FB_init : BOOL
VAR_INPUT
	bInitRetains : BOOL; // if TRUE, the retain variables are initialized (warm start / cold start)
	bInCopyCode : BOOL;  // if TRUE, the instance afterwards gets moved into the copy code (online change)
END_VAR
AddParameter('fScalar', fScalar);
AddInput('ipSrcImage', ipSrcImage);
AddInput('hrPrev', hrPrev);
AddOutput('ipDestImage', ipDestImage);
AddOutput('hresult',hresult);
END_METHOD

METHOD PROTECTED OnExecute
hresult.Value := F_VN_MultiplyImageWithScalar(
    fScalar := fScalar.Value,
    ipSrcImage := ipSrcImage.Value,
	ipDestImage := ipDestImage.Value,
	hrPrev:= hrPrev.Value);
END_METHOD

METHOD PUBLIC PreExecutionCheck
VAR_INPUT
	Check : I_PreExecutionChecks;
END_VAR
Check.IsTrue(ipSrcImage.IsValid, 'ipSrcImage must contain an image');
END_METHOD

END_FUNCTION_BLOCK

// ---- Nodes/Algebraic Image Ops/Node_F_VN_MultiplyImageWithVector.TcPOU
{attribute 'linkalways'} 
{attribute 'no_explicit_call' := 'This FB is a CLASS and must be accessed using methods or properties'}
{attribute 'enable_dynamic_creation'}
FUNCTION_BLOCK Node_F_VN_MultiplyImageWithVector EXTENDS VisionNode
VAR
    aVector : _TcVnVector4_LREAL;
    ipSrcImage : _ITcVnImage;
    ipDestImage : _ITcVnImage;
    hrPrev : _HRESULT(S_OK);
	hresult : _HRESULT(S_OK);
END_VAR

METHOD PUBLIC  Clone : I_Node
VAR
	pNode : POINTER TO Node_F_VN_MultiplyImageWithVector;
END_VAR
pNode := __NEW(Node_F_VN_MultiplyImageWithVector);
Clone := pNode^;
END_METHOD

METHOD FB_init : BOOL
VAR_INPUT
	bInitRetains : BOOL; // if TRUE, the retain variables are initialized (warm start / cold start)
	bInCopyCode : BOOL;  // if TRUE, the instance afterwards gets moved into the copy code (online change)
END_VAR
AddInput('aVector', aVector);
AddInput('ipSrcImage', ipSrcImage);
AddInput('hrPrev', hrPrev);
AddOutput('ipDestImage', ipDestImage);
AddOutput('hresult',hresult);
END_METHOD

METHOD PROTECTED OnExecute
hresult.Value := F_VN_MultiplyImageWithVector(
    aVector := aVector.Value,
    ipSrcImage := ipSrcImage.Value,
	ipDestImage := ipDestImage.Value,
	hrPrev:= hrPrev.Value);
END_METHOD

METHOD PUBLIC PreExecutionCheck
VAR_INPUT
	Check : I_PreExecutionChecks;
END_VAR
Check.IsTrue(ipSrcImage.IsValid, 'ipSrcImage must contain an image');
END_METHOD

END_FUNCTION_BLOCK

// ---- Nodes/Algebraic Image Ops/Node_F_VN_SubtractImageFromVector.TcPOU
{attribute 'linkalways'} 
{attribute 'no_explicit_call' := 'This FB is a CLASS and must be accessed using methods or properties'}
{attribute 'enable_dynamic_creation'}
FUNCTION_BLOCK Node_F_VN_SubtractImageFromVector EXTENDS VisionNode
VAR
    aVector : _TcVnVector4_LREAL;
    ipSrcImage : _ITcVnImage;
    ipDestImage : _ITcVnImage;
    hrPrev : _HRESULT(S_OK);
	hresult : _HRESULT(S_OK);
END_VAR

METHOD PUBLIC  Clone : I_Node
VAR
	pNode : POINTER TO Node_F_VN_SubtractImageFromVector;
END_VAR
pNode := __NEW(Node_F_VN_SubtractImageFromVector);
Clone := pNode^;
END_METHOD

METHOD FB_init : BOOL
VAR_INPUT
	bInitRetains : BOOL; // if TRUE, the retain variables are initialized (warm start / cold start)
	bInCopyCode : BOOL;  // if TRUE, the instance afterwards gets moved into the copy code (online change)
END_VAR
AddInput('aVector', aVector);
AddInput('ipSrcImage', ipSrcImage);
AddInput('hrPrev', hrPrev);
AddOutput('ipDestImage', ipDestImage);
AddOutput('hresult',hresult);
END_METHOD

METHOD PROTECTED OnExecute
hresult.Value := F_VN_SubtractImageFromVector(
    aVector := aVector.Value,
    ipSrcImage := ipSrcImage.Value,
	ipDestImage := ipDestImage.Value,
	hrPrev:= hrPrev.Value);
END_METHOD

METHOD PUBLIC PreExecutionCheck
VAR_INPUT
	Check : I_PreExecutionChecks;
END_VAR
Check.IsTrue(ipSrcImage.IsValid, 'ipSrcImage must contain an image');
END_METHOD

END_FUNCTION_BLOCK

// ---- Nodes/Algebraic Image Ops/Node_F_VN_SubtractScalarFromImage.TcPOU
{attribute 'linkalways'} 
{attribute 'no_explicit_call' := 'This FB is a CLASS and must be accessed using methods or properties'}
{attribute 'enable_dynamic_creation'}
FUNCTION_BLOCK Node_F_VN_SubtractScalarFromImage EXTENDS VisionNode
VAR
    ipSrcImage : _ITcVnImage;
    fScalar : _LREAL(0.0);
    ipDestImage : _ITcVnImage;
    hrPrev : _HRESULT(S_OK);
	hresult : _HRESULT(S_OK);
END_VAR

METHOD PUBLIC  Clone : I_Node
VAR
	pNode : POINTER TO Node_F_VN_SubtractScalarFromImage;
END_VAR
pNode := __NEW(Node_F_VN_SubtractScalarFromImage);
Clone := pNode^;
END_METHOD

METHOD FB_init : BOOL
VAR_INPUT
	bInitRetains : BOOL; // if TRUE, the retain variables are initialized (warm start / cold start)
	bInCopyCode : BOOL;  // if TRUE, the instance afterwards gets moved into the copy code (online change)
END_VAR
AddInput('ipSrcImage', ipSrcImage);
AddParameter('fScalar', fScalar);
AddInput('hrPrev', hrPrev);
AddOutput('ipDestImage', ipDestImage);
AddOutput('hresult',hresult);
END_METHOD

METHOD PROTECTED OnExecute
hresult.Value := F_VN_SubtractScalarFromImage(
    ipSrcImage := ipSrcImage.Value,
    fScalar := fScalar.Value,
	ipDestImage := ipDestImage.Value,
	hrPrev:= hrPrev.Value);
END_METHOD

METHOD PUBLIC PreExecutionCheck
VAR_INPUT
	Check : I_PreExecutionChecks;
END_VAR
Check.IsTrue(ipSrcImage.IsValid, 'ipSrcImage must contain an image');
END_METHOD

END_FUNCTION_BLOCK

// ---- Nodes/Algebraic Image Ops/Node_F_VN_MultiplyImages.TcPOU
{attribute 'linkalways'} 
{attribute 'no_explicit_call' := 'This FB is a CLASS and must be accessed using methods or properties'}
{attribute 'enable_dynamic_creation'}
FUNCTION_BLOCK Node_F_VN_MultiplyImages EXTENDS VisionNode
VAR
    ipSrcImage1 : _ITcVnImage;
    ipSrcImage2 : _ITcVnImage;
    ipDestImage : _ITcVnImage;
    hrPrev : _HRESULT(S_OK);
	hresult : _HRESULT(S_OK);
END_VAR

METHOD PUBLIC  Clone : I_Node
VAR
	pNode : POINTER TO Node_F_VN_MultiplyImages;
END_VAR
pNode := __NEW(Node_F_VN_MultiplyImages);
Clone := pNode^;
END_METHOD

METHOD FB_init : BOOL
VAR_INPUT
	bInitRetains : BOOL; // if TRUE, the retain variables are initialized (warm start / cold start)
	bInCopyCode : BOOL;  // if TRUE, the instance afterwards gets moved into the copy code (online change)
END_VAR
AddInput('ipSrcImage1', ipSrcImage1);
AddInput('ipSrcImage2', ipSrcImage2);
AddInput('hrPrev', hrPrev);
AddOutput('ipDestImage', ipDestImage);
AddOutput('hresult',hresult);
END_METHOD

METHOD PROTECTED OnExecute
hresult.Value := F_VN_MultiplyImages(
    ipSrcImage1 := ipSrcImage1.Value,
    ipSrcImage2 := ipSrcImage2.Value,
	ipDestImage := ipDestImage.Value,
	hrPrev:= hrPrev.Value);
END_METHOD

METHOD PUBLIC PreExecutionCheck
VAR_INPUT
	Check : I_PreExecutionChecks;
END_VAR
Check.IsTrue(ipSrcImage1.IsValid, 'ipSrcImage1 must contain an image');
Check.IsTrue(ipSrcImage2.IsValid, 'ipSrcImage2 must contain an image');
Check.IsTrue(IsImage1SizeEqualToImage2Size(ipSrcImage1.Value, ipSrcImage2.Value), 'ipSrcImage1 must be the same size as ipSrcImage2');
END_METHOD

END_FUNCTION_BLOCK

// ---- Nodes/Algebraic Image Ops/Node_F_VN_SubtractImages.TcPOU
{attribute 'linkalways'} 
{attribute 'no_explicit_call' := 'This FB is a CLASS and must be accessed using methods or properties'}
{attribute 'enable_dynamic_creation'}
FUNCTION_BLOCK Node_F_VN_SubtractImages EXTENDS VisionNode
VAR
    ipSrcImage1 : _ITcVnImage;
    ipSrcImage2 : _ITcVnImage;
    ipDestImage : _ITcVnImage;
    hrPrev : _HRESULT(S_OK);
	hresult : _HRESULT(S_OK);
END_VAR

METHOD PUBLIC  Clone : I_Node
VAR
	pNode : POINTER TO Node_F_VN_SubtractImages;
END_VAR
pNode := __NEW(Node_F_VN_SubtractImages);
Clone := pNode^;
END_METHOD

METHOD FB_init : BOOL
VAR_INPUT
	bInitRetains : BOOL; // if TRUE, the retain variables are initialized (warm start / cold start)
	bInCopyCode : BOOL;  // if TRUE, the instance afterwards gets moved into the copy code (online change)
END_VAR
AddInput('ipSrcImage1', ipSrcImage1);
AddInput('ipSrcImage2', ipSrcImage2);
AddInput('hrPrev', hrPrev);
AddOutput('ipDestImage', ipDestImage);
AddOutput('hresult',hresult);
END_METHOD

METHOD PROTECTED OnExecute
hresult.Value := F_VN_SubtractImages(
    ipSrcImage1 := ipSrcImage1.Value,
    ipSrcImage2 := ipSrcImage2.Value,
	ipDestImage := ipDestImage.Value,
	hrPrev:= hrPrev.Value);
END_METHOD

METHOD PUBLIC PreExecutionCheck
VAR_INPUT
	Check : I_PreExecutionChecks;
END_VAR
Check.IsTrue(ipSrcImage1.IsValid, 'ipSrcImage1 must contain an image');
Check.IsTrue(ipSrcImage2.IsValid, 'ipSrcImage2 must contain an image');
Check.IsTrue(IsImage1SizeEqualToImage2Size(ipSrcImage1.Value, ipSrcImage2.Value), 'ipSrcImage1 must be the same size as ipSrcImage2');
END_METHOD

END_FUNCTION_BLOCK

// ---- Nodes/Algebraic Image Ops/Node_F_VN_MaxImage.TcPOU
{attribute 'linkalways'} 
{attribute 'no_explicit_call' := 'This FB is a CLASS and must be accessed using methods or properties'}
{attribute 'enable_dynamic_creation'}
FUNCTION_BLOCK Node_F_VN_MaxImage EXTENDS VisionNode
VAR
    ipSrcImage1 : _ITcVnImage;
    ipSrcImage2 : _ITcVnImage;
    ipDestImage : _ITcVnImage;
    hrPrev : _HRESULT(S_OK);
	hresult : _HRESULT(S_OK);
END_VAR

METHOD PUBLIC  Clone : I_Node
VAR
	pNode : POINTER TO Node_F_VN_MaxImage;
END_VAR
pNode := __NEW(Node_F_VN_MaxImage);
Clone := pNode^;
END_METHOD

METHOD FB_init : BOOL
VAR_INPUT
	bInitRetains : BOOL; // if TRUE, the retain variables are initialized (warm start / cold start)
	bInCopyCode : BOOL;  // if TRUE, the instance afterwards gets moved into the copy code (online change)
END_VAR
AddInput('ipSrcImage1', ipSrcImage1);
AddInput('ipSrcImage2', ipSrcImage2);
AddInput('hrPrev', hrPrev);
AddOutput('ipDestImage', ipDestImage);
AddOutput('hresult',hresult);
END_METHOD

METHOD PROTECTED OnExecute
hresult.Value := F_VN_MaxImage(
    ipSrcImage1 := ipSrcImage1.Value,
    ipSrcImage2 := ipSrcImage2.Value,
	ipDestImage := ipDestImage.Value,
	hrPrev:= hrPrev.Value);
END_METHOD

METHOD PUBLIC PreExecutionCheck
VAR_INPUT
	Check : I_PreExecutionChecks;
END_VAR
Check.IsTrue(ipSrcImage1.IsValid, 'ipSrcImage1 must contain an image');
Check.IsTrue(ipSrcImage2.IsValid, 'ipSrcImage2 must contain an image');
Check.IsTrue(IsImage1SizeEqualToImage2Size(ipSrcImage1.Value, ipSrcImage2.Value), 'ipSrcImage1 must be the same size as ipSrcImage2');
END_METHOD

END_FUNCTION_BLOCK

// ---- Nodes/Algebraic Image Ops/Node_F_VN_BitwiseOrImages.TcPOU
{attribute 'linkalways'} 
{attribute 'no_explicit_call' := 'This FB is a CLASS and must be accessed using methods or properties'}
{attribute 'enable_dynamic_creation'}
FUNCTION_BLOCK Node_F_VN_BitwiseOrImages EXTENDS VisionNode
VAR
    ipSrcImage1 : _ITcVnImage;
    ipSrcImage2 : _ITcVnImage;
    ipDestImage : _ITcVnImage;
    hrPrev : _HRESULT(S_OK);
	hresult : _HRESULT(S_OK);
END_VAR

METHOD PUBLIC  Clone : I_Node
VAR
	pNode : POINTER TO Node_F_VN_BitwiseOrImages;
END_VAR
pNode := __NEW(Node_F_VN_BitwiseOrImages);
Clone := pNode^;
END_METHOD

METHOD FB_init : BOOL
VAR_INPUT
	bInitRetains : BOOL; // if TRUE, the retain variables are initialized (warm start / cold start)
	bInCopyCode : BOOL;  // if TRUE, the instance afterwards gets moved into the copy code (online change)
END_VAR
AddInput('ipSrcImage1', ipSrcImage1);
AddInput('ipSrcImage2', ipSrcImage2);
AddInput('hrPrev', hrPrev);
AddOutput('ipDestImage', ipDestImage);
AddOutput('hresult',hresult);
END_METHOD

METHOD PROTECTED OnExecute
hresult.Value := F_VN_BitwiseOrImages(
    ipSrcImage1 := ipSrcImage1.Value,
    ipSrcImage2 := ipSrcImage2.Value,
	ipDestImage := ipDestImage.Value,
	hrPrev:= hrPrev.Value);
END_METHOD

METHOD PUBLIC PreExecutionCheck
VAR_INPUT
	Check : I_PreExecutionChecks;
END_VAR
Check.IsTrue(ipSrcImage1.IsValid, 'ipSrcImage1 must contain an image');
Check.IsTrue(ipSrcImage2.IsValid, 'ipSrcImage2 must contain an image');
Check.IsTrue(IsImage1SizeEqualToImage2Size(ipSrcImage1.Value, ipSrcImage2.Value), 'ipSrcImage1 must be the same size as ipSrcImage2');
END_METHOD

END_FUNCTION_BLOCK

// ---- Nodes/Algebraic Image Ops/Node_F_VN_BitwiseNotImage.TcPOU
{attribute 'linkalways'} 
{attribute 'no_explicit_call' := 'This FB is a CLASS and must be accessed using methods or properties'}
{attribute 'enable_dynamic_creation'}
FUNCTION_BLOCK Node_F_VN_BitwiseNotImage EXTENDS VisionNode
VAR
    ipSrcImage : _ITcVnImage;
    ipDestImage : _ITcVnImage;
    hrPrev : _HRESULT(S_OK);
	hresult : _HRESULT(S_OK);
END_VAR

METHOD PUBLIC  Clone : I_Node
VAR
	pNode : POINTER TO Node_F_VN_BitwiseNotImage;
END_VAR
pNode := __NEW(Node_F_VN_BitwiseNotImage);
Clone := pNode^;
END_METHOD

METHOD FB_init : BOOL
VAR_INPUT
	bInitRetains : BOOL; // if TRUE, the retain variables are initialized (warm start / cold start)
	bInCopyCode : BOOL;  // if TRUE, the instance afterwards gets moved into the copy code (online change)
END_VAR
AddInput('ipSrcImage', ipSrcImage);
AddInput('hrPrev', hrPrev);
AddOutput('ipDestImage', ipDestImage);
AddOutput('hresult',hresult);
END_METHOD

METHOD PROTECTED OnExecute
hresult.Value := F_VN_BitwiseNotImage(
    ipSrcImage := ipSrcImage.Value,
	ipDestImage := ipDestImage.Value,
	hrPrev:= hrPrev.Value);
END_METHOD

METHOD PUBLIC PreExecutionCheck
VAR_INPUT
	Check : I_PreExecutionChecks;
END_VAR
Check.IsTrue(ipSrcImage.IsValid, 'ipSrcImage must contain an image');
END_METHOD

END_FUNCTION_BLOCK

// ---- Nodes/Algebraic Image Ops/Node_F_VN_BitwiseAndImages.TcPOU
{attribute 'linkalways'} 
{attribute 'no_explicit_call' := 'This FB is a CLASS and must be accessed using methods or properties'}
{attribute 'enable_dynamic_creation'}
FUNCTION_BLOCK Node_F_VN_BitwiseAndImages EXTENDS VisionNode
VAR
    ipSrcImage1 : _ITcVnImage;
    ipSrcImage2 : _ITcVnImage;
    ipDestImage : _ITcVnImage;
    hrPrev : _HRESULT(S_OK);
	hresult : _HRESULT(S_OK);
END_VAR

METHOD PUBLIC  Clone : I_Node
VAR
	pNode : POINTER TO Node_F_VN_BitwiseAndImages;
END_VAR
pNode := __NEW(Node_F_VN_BitwiseAndImages);
Clone := pNode^;
END_METHOD

METHOD FB_init : BOOL
VAR_INPUT
	bInitRetains : BOOL; // if TRUE, the retain variables are initialized (warm start / cold start)
	bInCopyCode : BOOL;  // if TRUE, the instance afterwards gets moved into the copy code (online change)
END_VAR
AddInput('ipSrcImage1', ipSrcImage1);
AddInput('ipSrcImage2', ipSrcImage2);
AddInput('hrPrev', hrPrev);
AddOutput('ipDestImage', ipDestImage);
AddOutput('hresult',hresult);
END_METHOD

METHOD PROTECTED OnExecute
hresult.Value := F_VN_BitwiseAndImages(
    ipSrcImage1 := ipSrcImage1.Value,
    ipSrcImage2 := ipSrcImage2.Value,
	ipDestImage := ipDestImage.Value,
	hrPrev:= hrPrev.Value);
END_METHOD

METHOD PUBLIC PreExecutionCheck
VAR_INPUT
	Check : I_PreExecutionChecks;
END_VAR
Check.IsTrue(ipSrcImage1.IsValid, 'ipSrcImage1 must contain an image');
Check.IsTrue(ipSrcImage2.IsValid, 'ipSrcImage2 must contain an image');
Check.IsTrue(IsImage1SizeEqualToImage2Size(ipSrcImage1.Value, ipSrcImage2.Value), 'ipSrcImage1 must be the same size as ipSrcImage2');
END_METHOD

END_FUNCTION_BLOCK

// ---- Nodes/Algebraic Image Ops/Node_F_VN_BitwiseXorImages.TcPOU
{attribute 'linkalways'} 
{attribute 'no_explicit_call' := 'This FB is a CLASS and must be accessed using methods or properties'}
{attribute 'enable_dynamic_creation'}
FUNCTION_BLOCK Node_F_VN_BitwiseXorImages EXTENDS VisionNode
VAR
    ipSrcImage1 : _ITcVnImage;
    ipSrcImage2 : _ITcVnImage;
    ipDestImage : _ITcVnImage;
    hrPrev : _HRESULT(S_OK);
	hresult : _HRESULT(S_OK);
END_VAR

METHOD PUBLIC  Clone : I_Node
VAR
	pNode : POINTER TO Node_F_VN_BitwiseXorImages;
END_VAR
pNode := __NEW(Node_F_VN_BitwiseXorImages);
Clone := pNode^;
END_METHOD

METHOD FB_init : BOOL
VAR_INPUT
	bInitRetains : BOOL; // if TRUE, the retain variables are initialized (warm start / cold start)
	bInCopyCode : BOOL;  // if TRUE, the instance afterwards gets moved into the copy code (online change)
END_VAR
AddInput('ipSrcImage1', ipSrcImage1);
AddInput('ipSrcImage2', ipSrcImage2);
AddInput('hrPrev', hrPrev);
AddOutput('ipDestImage', ipDestImage);
AddOutput('hresult',hresult);
END_METHOD

METHOD PROTECTED OnExecute
hresult.Value := F_VN_BitwiseXorImages(
    ipSrcImage1 := ipSrcImage1.Value,
    ipSrcImage2 := ipSrcImage2.Value,
	ipDestImage := ipDestImage.Value,
	hrPrev:= hrPrev.Value);
END_METHOD

METHOD PUBLIC PreExecutionCheck
VAR_INPUT
	Check : I_PreExecutionChecks;
END_VAR
Check.IsTrue(ipSrcImage1.IsValid, 'ipSrcImage1 must contain an image');
Check.IsTrue(ipSrcImage2.IsValid, 'ipSrcImage2 must contain an image');
Check.IsTrue(IsImage1SizeEqualToImage2Size(ipSrcImage1.Value, ipSrcImage2.Value), 'ipSrcImage1 must be the same size as ipSrcImage2');
END_METHOD

END_FUNCTION_BLOCK

// ---- Nodes/Algebraic Image Ops/Node_F_VN_MinImage.TcPOU
{attribute 'linkalways'} 
{attribute 'no_explicit_call' := 'This FB is a CLASS and must be accessed using methods or properties'}
{attribute 'enable_dynamic_creation'}
FUNCTION_BLOCK Node_F_VN_MinImage EXTENDS VisionNode
VAR
    ipSrcImage1 : _ITcVnImage;
    ipSrcImage2 : _ITcVnImage;
    ipDestImage : _ITcVnImage;
    hrPrev : _HRESULT(S_OK);
	hresult : _HRESULT(S_OK);
END_VAR

METHOD PUBLIC  Clone : I_Node
VAR
	pNode : POINTER TO Node_F_VN_MinImage;
END_VAR
pNode := __NEW(Node_F_VN_MinImage);
Clone := pNode^;
END_METHOD

METHOD FB_init : BOOL
VAR_INPUT
	bInitRetains : BOOL; // if TRUE, the retain variables are initialized (warm start / cold start)
	bInCopyCode : BOOL;  // if TRUE, the instance afterwards gets moved into the copy code (online change)
END_VAR
AddInput('ipSrcImage1', ipSrcImage1);
AddInput('ipSrcImage2', ipSrcImage2);
AddInput('hrPrev', hrPrev);
AddOutput('ipDestImage', ipDestImage);
AddOutput('hresult',hresult);
END_METHOD

METHOD PROTECTED OnExecute
hresult.Value := F_VN_MinImage(
    ipSrcImage1 := ipSrcImage1.Value,
    ipSrcImage2 := ipSrcImage2.Value,
	ipDestImage := ipDestImage.Value,
	hrPrev:= hrPrev.Value);
END_METHOD

METHOD PUBLIC PreExecutionCheck
VAR_INPUT
	Check : I_PreExecutionChecks;
END_VAR
Check.IsTrue(ipSrcImage1.IsValid, 'ipSrcImage1 must contain an image');
Check.IsTrue(ipSrcImage2.IsValid, 'ipSrcImage2 must contain an image');
Check.IsTrue(IsImage1SizeEqualToImage2Size(ipSrcImage1.Value, ipSrcImage2.Value), 'ipSrcImage1 must be the same size as ipSrcImage2');
END_METHOD

END_FUNCTION_BLOCK

// ---- Nodes/Algebraic Image Ops/Node_F_VN_DivideImages.TcPOU
{attribute 'linkalways'} 
{attribute 'no_explicit_call' := 'This FB is a CLASS and must be accessed using methods or properties'}
{attribute 'enable_dynamic_creation'}
FUNCTION_BLOCK Node_F_VN_DivideImages EXTENDS VisionNode
VAR
    ipSrcImage1 : _ITcVnImage;
    ipSrcImage2 : _ITcVnImage;
    ipDestImage : _ITcVnImage;
    hrPrev : _HRESULT(S_OK);
	hresult : _HRESULT(S_OK);
END_VAR

METHOD PUBLIC  Clone : I_Node
VAR
	pNode : POINTER TO Node_F_VN_DivideImages;
END_VAR
pNode := __NEW(Node_F_VN_DivideImages);
Clone := pNode^;
END_METHOD

METHOD FB_init : BOOL
VAR_INPUT
	bInitRetains : BOOL; // if TRUE, the retain variables are initialized (warm start / cold start)
	bInCopyCode : BOOL;  // if TRUE, the instance afterwards gets moved into the copy code (online change)
END_VAR
AddInput('ipSrcImage1', ipSrcImage1);
AddInput('ipSrcImage2', ipSrcImage2);
AddInput('hrPrev', hrPrev);
AddOutput('ipDestImage', ipDestImage);
AddOutput('hresult',hresult);
END_METHOD

METHOD PROTECTED OnExecute
hresult.Value := F_VN_DivideImages(
    ipSrcImage1 := ipSrcImage1.Value,
    ipSrcImage2 := ipSrcImage2.Value,
	ipDestImage := ipDestImage.Value,
	hrPrev:= hrPrev.Value);
END_METHOD

METHOD PUBLIC PreExecutionCheck
VAR_INPUT
	Check : I_PreExecutionChecks;
END_VAR
Check.IsTrue(ipSrcImage1.IsValid, 'ipSrcImage1 must contain an image');
Check.IsTrue(ipSrcImage2.IsValid, 'ipSrcImage2 must contain an image');
Check.IsTrue(IsImage1SizeEqualToImage2Size(ipSrcImage1.Value, ipSrcImage2.Value), 'ipSrcImage1 must be the same size as ipSrcImage2');
END_METHOD

END_FUNCTION_BLOCK

// ---- Nodes/Algebraic Image Ops/Node_F_VN_SubtractImageFromScalar.TcPOU
{attribute 'linkalways'} 
{attribute 'no_explicit_call' := 'This FB is a CLASS and must be accessed using methods or properties'}
{attribute 'enable_dynamic_creation'}
FUNCTION_BLOCK Node_F_VN_SubtractImageFromScalar EXTENDS VisionNode
VAR
    fScalar : _LREAL(0.0);
    ipSrcImage : _ITcVnImage;
    ipDestImage : _ITcVnImage;
    hrPrev : _HRESULT(S_OK);
	hresult : _HRESULT(S_OK);
END_VAR

METHOD PUBLIC  Clone : I_Node
VAR
	pNode : POINTER TO Node_F_VN_SubtractImageFromScalar;
END_VAR
pNode := __NEW(Node_F_VN_SubtractImageFromScalar);
Clone := pNode^;
END_METHOD

METHOD FB_init : BOOL
VAR_INPUT
	bInitRetains : BOOL; // if TRUE, the retain variables are initialized (warm start / cold start)
	bInCopyCode : BOOL;  // if TRUE, the instance afterwards gets moved into the copy code (online change)
END_VAR
AddParameter('fScalar', fScalar);
AddInput('ipSrcImage', ipSrcImage);
AddInput('hrPrev', hrPrev);
AddOutput('ipDestImage', ipDestImage);
AddOutput('hresult',hresult);
END_METHOD

METHOD PROTECTED OnExecute
hresult.Value := F_VN_SubtractImageFromScalar(
    fScalar := fScalar.Value,
    ipSrcImage := ipSrcImage.Value,
	ipDestImage := ipDestImage.Value,
	hrPrev:= hrPrev.Value);
END_METHOD

METHOD PUBLIC PreExecutionCheck
VAR_INPUT
	Check : I_PreExecutionChecks;
END_VAR
Check.IsTrue(ipSrcImage.IsValid, 'ipSrcImage must contain an image');
END_METHOD

END_FUNCTION_BLOCK

// ---- Nodes/Algebraic Image Ops/Node_F_VN_AddScalarToImage.TcPOU
{attribute 'linkalways'} 
{attribute 'no_explicit_call' := 'This FB is a CLASS and must be accessed using methods or properties'}
{attribute 'enable_dynamic_creation'}
FUNCTION_BLOCK Node_F_VN_AddScalarToImage EXTENDS VisionNode
VAR
    fScalar : _LREAL(0.0);
    ipSrcImage : _ITcVnImage;
    ipDestImage : _ITcVnImage;
    hrPrev : _HRESULT(S_OK);
	hresult : _HRESULT(S_OK);
END_VAR

METHOD PUBLIC  Clone : I_Node
VAR
	pNode : POINTER TO Node_F_VN_AddScalarToImage;
END_VAR
pNode := __NEW(Node_F_VN_AddScalarToImage);
Clone := pNode^;
END_METHOD

METHOD FB_init : BOOL
VAR_INPUT
	bInitRetains : BOOL; // if TRUE, the retain variables are initialized (warm start / cold start)
	bInCopyCode : BOOL;  // if TRUE, the instance afterwards gets moved into the copy code (online change)
END_VAR
AddParameter('fScalar', fScalar);
AddInput('ipSrcImage', ipSrcImage);
AddInput('hrPrev', hrPrev);
AddOutput('ipDestImage', ipDestImage);
AddOutput('hresult',hresult);
END_METHOD

METHOD PROTECTED OnExecute
hresult.Value := F_VN_AddScalarToImage(
    fScalar := fScalar.Value,
    ipSrcImage := ipSrcImage.Value,
	ipDestImage := ipDestImage.Value,
	hrPrev:= hrPrev.Value);
END_METHOD

METHOD PUBLIC PreExecutionCheck
VAR_INPUT
	Check : I_PreExecutionChecks;
END_VAR
Check.IsTrue(ipSrcImage.IsValid, 'ipSrcImage must contain an image');
END_METHOD

END_FUNCTION_BLOCK

// ---- Nodes/Algebraic Image Ops/Node_F_VN_SubtractVectorFromImage.TcPOU
{attribute 'linkalways'} 
{attribute 'no_explicit_call' := 'This FB is a CLASS and must be accessed using methods or properties'}
{attribute 'enable_dynamic_creation'}
FUNCTION_BLOCK Node_F_VN_SubtractVectorFromImage EXTENDS VisionNode
VAR
    ipSrcImage : _ITcVnImage;
    aVector : _TcVnVector4_LREAL;
    ipDestImage : _ITcVnImage;
    hrPrev : _HRESULT(S_OK);
	hresult : _HRESULT(S_OK);
END_VAR

METHOD PUBLIC  Clone : I_Node
VAR
	pNode : POINTER TO Node_F_VN_SubtractVectorFromImage;
END_VAR
pNode := __NEW(Node_F_VN_SubtractVectorFromImage);
Clone := pNode^;
END_METHOD

METHOD FB_init : BOOL
VAR_INPUT
	bInitRetains : BOOL; // if TRUE, the retain variables are initialized (warm start / cold start)
	bInCopyCode : BOOL;  // if TRUE, the instance afterwards gets moved into the copy code (online change)
END_VAR
AddInput('ipSrcImage', ipSrcImage);
AddInput('aVector', aVector);
AddInput('hrPrev', hrPrev);
AddOutput('ipDestImage', ipDestImage);
AddOutput('hresult',hresult);
END_METHOD

METHOD PROTECTED OnExecute
hresult.Value := F_VN_SubtractVectorFromImage(
    ipSrcImage := ipSrcImage.Value,
    aVector := aVector.Value,
	ipDestImage := ipDestImage.Value,
	hrPrev:= hrPrev.Value);
END_METHOD

METHOD PUBLIC PreExecutionCheck
VAR_INPUT
	Check : I_PreExecutionChecks;
END_VAR
Check.IsTrue(ipSrcImage.IsValid, 'ipSrcImage must contain an image');
END_METHOD

END_FUNCTION_BLOCK

// ---- Nodes/Basic Container Ops/Node_F_VN_CreateContainer.TcPOU
{attribute 'linkalways'} 
{attribute 'no_explicit_call' := 'This FB is a CLASS and must be accessed using methods or properties'}
{attribute 'enable_dynamic_creation'}
FUNCTION_BLOCK Node_F_VN_CreateContainer EXTENDS VisionNode
VAR
    ipContainer : _ITcVnContainer;
    nTypeGuid : _GUID();
    nElementNum : _ULINT(1);
    hrPrev : _HRESULT(S_OK);
	hresult : _HRESULT(S_OK);
END_VAR

METHOD PUBLIC  Clone : I_Node
VAR
	pNode : POINTER TO Node_F_VN_CreateContainer;
END_VAR
pNode := __NEW(Node_F_VN_CreateContainer);
Clone := pNode^;
END_METHOD

METHOD FB_init : BOOL
VAR_INPUT
	bInitRetains : BOOL; // if TRUE, the retain variables are initialized (warm start / cold start)
	bInCopyCode : BOOL;  // if TRUE, the instance afterwards gets moved into the copy code (online change)
END_VAR
AddParameter('nTypeGuid', nTypeGuid);
AddParameter('nElementNum', nElementNum);
AddInput('hrPrev', hrPrev);
AddOutput('ipContainer', ipContainer);
AddOutput('hresult',hresult);
END_METHOD

METHOD PROTECTED OnExecute
hresult.Value := F_VN_CreateContainer(
    ipContainer := ipContainer.Value,
    nTypeGuid := nTypeGuid.Value,
    nElementNum := nElementNum.Value,
	hrPrev:= hrPrev.Value);
END_METHOD

METHOD PUBLIC PreExecutionCheck
VAR_INPUT
	Check : I_PreExecutionChecks;
END_VAR
VAR
	typeGuid : GUID;
	match : BOOL;
END_VAR
Check.IsTrue((nElementNum.Value >= 0), 'nElementNum must be greater than or equal to 0');

match := 
    nTypeGuid.EqualsGuid(ContainerType_Vector_SINT) OR_ELSE
    nTypeGuid.EqualsGuid(ContainerType_Vector_USINT) OR_ELSE
    nTypeGuid.EqualsGuid(ContainerType_Vector_INT) OR_ELSE
    nTypeGuid.EqualsGuid(ContainerType_Vector_UINT) OR_ELSE
    nTypeGuid.EqualsGuid(ContainerType_Vector_DINT) OR_ELSE
    nTypeGuid.EqualsGuid(ContainerType_Vector_UDINT) OR_ELSE
    nTypeGuid.EqualsGuid(ContainerType_Vector_ULINT) OR_ELSE
    nTypeGuid.EqualsGuid(ContainerType_Vector_REAL) OR_ELSE
    nTypeGuid.EqualsGuid(ContainerType_Vector_LREAL) OR_ELSE
    nTypeGuid.EqualsGuid(ContainerType_Vector_ITcVnImage) OR_ELSE
    nTypeGuid.EqualsGuid(ContainerType_Vector_TcVnPoint2_DINT) OR_ELSE
    nTypeGuid.EqualsGuid(ContainerType_Vector_TcVnPoint2_REAL) OR_ELSE
    nTypeGuid.EqualsGuid(ContainerType_Vector_TcVnPoint2_LREAL) OR_ELSE
    nTypeGuid.EqualsGuid(ContainerType_Vector_TcVnPoint3_REAL) OR_ELSE
    nTypeGuid.EqualsGuid(ContainerType_Vector_TcVnPoint3_LREAL) OR_ELSE
    nTypeGuid.EqualsGuid(ContainerType_Vector_Vector_TcVnPoint2_DINT) OR_ELSE
    nTypeGuid.EqualsGuid(ContainerType_Vector_Vector_TcVnPoint2_REAL) OR_ELSE
    nTypeGuid.EqualsGuid(ContainerType_Vector_Vector_TcVnPoint3_REAL) OR_ELSE
    nTypeGuid.EqualsGuid(ContainerType_Vector_Vector_UDINT) OR_ELSE
    nTypeGuid.EqualsGuid(ContainerType_Vector_Vector_ULINT) OR_ELSE
    nTypeGuid.EqualsGuid(ContainerType_Vector_Vector_REAL) OR_ELSE
    nTypeGuid.EqualsGuid(ContainerType_Vector_Vector_LREAL) OR_ELSE
    nTypeGuid.EqualsGuid(ContainerType_Vector_TcVnVector2_SINT) OR_ELSE
    nTypeGuid.EqualsGuid(ContainerType_Vector_TcVnVector2_USINT) OR_ELSE
    nTypeGuid.EqualsGuid(ContainerType_Vector_TcVnVector2_INT) OR_ELSE
    nTypeGuid.EqualsGuid(ContainerType_Vector_TcVnVector2_UINT) OR_ELSE
    nTypeGuid.EqualsGuid(ContainerType_Vector_TcVnVector2_DINT) OR_ELSE
    nTypeGuid.EqualsGuid(ContainerType_Vector_TcVnVector2_REAL) OR_ELSE
    nTypeGuid.EqualsGuid(ContainerType_Vector_TcVnVector3_SINT) OR_ELSE
    nTypeGuid.EqualsGuid(ContainerType_Vector_TcVnVector3_USINT) OR_ELSE
    nTypeGuid.EqualsGuid(ContainerType_Vector_TcVnVector3_INT) OR_ELSE
    nTypeGuid.EqualsGuid(ContainerType_Vector_TcVnVector3_UINT) OR_ELSE
    nTypeGuid.EqualsGuid(ContainerType_Vector_TcVnVector3_REAL) OR_ELSE
    nTypeGuid.EqualsGuid(ContainerType_Vector_TcVnVector4_SINT) OR_ELSE
    nTypeGuid.EqualsGuid(ContainerType_Vector_TcVnVector4_USINT) OR_ELSE
    nTypeGuid.EqualsGuid(ContainerType_Vector_TcVnVector4_INT) OR_ELSE
    nTypeGuid.EqualsGuid(ContainerType_Vector_TcVnVector4_UINT) OR_ELSE
    nTypeGuid.EqualsGuid(ContainerType_Vector_TcVnVector4_DINT) OR_ELSE
    nTypeGuid.EqualsGuid(ContainerType_Vector_TcVnVector4_REAL) OR_ELSE
    nTypeGuid.EqualsGuid(ContainerType_Vector_TcVnVector4_LREAL) OR_ELSE
    nTypeGuid.EqualsGuid(ContainerType_Vector_TcVnRectangle_DINT) OR_ELSE
    nTypeGuid.EqualsGuid(ContainerType_Vector_TcVnRotatedRectangle) OR_ELSE
    nTypeGuid.EqualsGuid(ContainerType_Vector_TcVnKeyPoint) OR_ELSE
    nTypeGuid.EqualsGuid(ContainerType_Vector_TcVnDMatch) OR_ELSE
    nTypeGuid.EqualsGuid(ContainerType_Vector_Vector_TcVnDMatch) OR_ELSE
    nTypeGuid.EqualsGuid(ContainerType_String_SINT) OR_ELSE
    nTypeGuid.EqualsGuid(ContainerType_Vector_String_SINT);
	
Check.IsTrue(match, 'nTypeGuid must be a valid GUID for containers');
END_METHOD

END_FUNCTION_BLOCK

// ---- Nodes/Basic Container Ops/Node_F_VN_ExportContainer_String.TcPOU
{attribute 'linkalways'} 
{attribute 'no_explicit_call' := 'This FB is a CLASS and must be accessed using methods or properties'}
{attribute 'enable_dynamic_creation'}
FUNCTION_BLOCK Node_F_VN_ExportContainer_String EXTENDS VisionNode
VAR
    ipContainer : _ITcVnContainer;
    sText : _STRING('');
    nMaxLength : _ULINT(0);
    hrPrev : _HRESULT(S_OK);
	hresult : _HRESULT(S_OK);
END_VAR

METHOD PUBLIC  Clone : I_Node
VAR
	pNode : POINTER TO Node_F_VN_ExportContainer_String;
END_VAR
pNode := __NEW(Node_F_VN_ExportContainer_String);
Clone := pNode^;
END_METHOD

METHOD FB_init : BOOL
VAR_INPUT
	bInitRetains : BOOL; // if TRUE, the retain variables are initialized (warm start / cold start)
	bInCopyCode : BOOL;  // if TRUE, the instance afterwards gets moved into the copy code (online change)
END_VAR
AddInput('ipContainer', ipContainer);
AddParameter('nMaxLength', nMaxLength);
AddInput('hrPrev', hrPrev);
AddOutput('sText', sText);
AddOutput('hresult',hresult);
END_METHOD

METHOD PROTECTED OnExecute
hresult.Value := F_VN_ExportContainer_String(
	ipContainer := ipContainer.Value,
    sText := sText.Value,
    nMaxLength := nMaxLength.Value,
	hrPrev:= hrPrev.Value);
END_METHOD

METHOD PUBLIC PreExecutionCheck
VAR_INPUT
	Check : I_PreExecutionChecks;
END_VAR
Check.IsTrue(ipContainer.IsValid, 'ipContainer must be a valid container');
Check.IsTrue(ipContainer.IsType(TC_GLOBAL_CONST_LIST.ContainerType_String_SINT), 'ipContainer contains incorrect type');
END_METHOD

END_FUNCTION_BLOCK

// ---- Nodes/Basic Container Ops/Node_F_VN_ExtractContainerRange.TcPOU
{attribute 'linkalways'} 
{attribute 'no_explicit_call' := 'This FB is a CLASS and must be accessed using methods or properties'}
{attribute 'enable_dynamic_creation'}
FUNCTION_BLOCK Node_F_VN_ExtractContainerRange EXTENDS VisionNode
VAR
    ipSrcContainer : _ITcVnContainer;
    ipDestContainer : _ITcVnContainer;
    nFirstIdx : _ULINT(0);
    nLastIdx : _ULINT(0);
    hrPrev : _HRESULT(S_OK);
	hresult : _HRESULT(S_OK);
END_VAR

METHOD PUBLIC  Clone : I_Node
VAR
	pNode : POINTER TO Node_F_VN_ExtractContainerRange;
END_VAR
pNode := __NEW(Node_F_VN_ExtractContainerRange);
Clone := pNode^;
END_METHOD

METHOD FB_init : BOOL
VAR_INPUT
	bInitRetains : BOOL; // if TRUE, the retain variables are initialized (warm start / cold start)
	bInCopyCode : BOOL;  // if TRUE, the instance afterwards gets moved into the copy code (online change)
END_VAR
AddInput('ipSrcContainer', ipSrcContainer);
AddParameter('nFirstIdx', nFirstIdx);
AddParameter('nLastIdx', nLastIdx);
AddInput('hrPrev', hrPrev);
AddOutput('ipDestContainer', ipDestContainer);
AddOutput('hresult',hresult);
END_METHOD

METHOD PROTECTED OnExecute
hresult.Value := F_VN_ExtractContainerRange(
	ipSrcContainer := ipSrcContainer.Value,
    ipDestContainer := ipDestContainer.Value,
    nFirstIdx := nFirstIdx.Value,
    nLastIdx := nLastIdx.Value,
	hrPrev:= hrPrev.Value);
END_METHOD

METHOD PUBLIC PreExecutionCheck
VAR_INPUT
	Check : I_PreExecutionChecks;
END_VAR
VAR
    empty : BOOL;
    elementNum : ULINT;
END_VAR
Check.IsTrue(ipSrcContainer.IsValid, 'ipSrcContainer must be a valid container');
Check.IsTrue(ipSrcContainer.TryGetElementNum(elementNum) AND (elementNum > 0), 'ipSrcContainer must not be empty');
Check.IsTrue(nLastIdx.Value >= nFirstIdx.Value, 'nLastIdx must be greater than or equal to nFirstIdx');
Check.IsTrue((nLastIdx.Value <= (elementNum - 1)), 'nLastIdx out of range');
END_METHOD

END_FUNCTION_BLOCK

// ---- Nodes/Basic Container Ops/Node_F_VN_ReverseContainer.TcPOU
{attribute 'linkalways'} 
{attribute 'no_explicit_call' := 'This FB is a CLASS and must be accessed using methods or properties'}
{attribute 'enable_dynamic_creation'}
FUNCTION_BLOCK Node_F_VN_ReverseContainer EXTENDS VisionNode
VAR
    ipContainer : _ITcVnContainer;
    hrPrev : _HRESULT(S_OK);
	hresult : _HRESULT(S_OK);
END_VAR

METHOD PUBLIC  Clone : I_Node
VAR
	pNode : POINTER TO Node_F_VN_ReverseContainer;
END_VAR
pNode := __NEW(Node_F_VN_ReverseContainer);
Clone := pNode^;
END_METHOD

METHOD FB_init : BOOL
VAR_INPUT
	bInitRetains : BOOL; // if TRUE, the retain variables are initialized (warm start / cold start)
	bInCopyCode : BOOL;  // if TRUE, the instance afterwards gets moved into the copy code (online change)
END_VAR
AddInput('ipContainer', ipContainer);
AddInput('hrPrev', hrPrev);
AddOutput('hresult',hresult);
END_METHOD

METHOD PROTECTED OnExecute
hresult.Value := F_VN_ReverseContainer(
	ipContainer := ipContainer.Value,
	hrPrev:= hrPrev.Value);
END_METHOD

METHOD PUBLIC PreExecutionCheck
VAR_INPUT
	Check : I_PreExecutionChecks;
END_VAR
Check.IsTrue(ipContainer.IsValid, 'ipContainer must be a valid container');
END_METHOD

END_FUNCTION_BLOCK

// ---- Nodes/Basic Container Ops/Node_F_VN_GetNumberOfElements.TcPOU
{attribute 'linkalways'} 
{attribute 'no_explicit_call' := 'This FB is a CLASS and must be accessed using methods or properties'}
{attribute 'enable_dynamic_creation'}
FUNCTION_BLOCK Node_F_VN_GetNumberOfElements EXTENDS VisionNode
VAR
    ipContainer : _ITcVnContainer;
    nNumberOfElements : _ULINT(0);
    hrPrev : _HRESULT(S_OK);
	hresult : _HRESULT(S_OK);
END_VAR

METHOD PUBLIC  Clone : I_Node
VAR
	pNode : POINTER TO Node_F_VN_GetNumberOfElements;
END_VAR
pNode := __NEW(Node_F_VN_GetNumberOfElements);
Clone := pNode^;
END_METHOD

METHOD FB_init : BOOL
VAR_INPUT
	bInitRetains : BOOL; // if TRUE, the retain variables are initialized (warm start / cold start)
	bInCopyCode : BOOL;  // if TRUE, the instance afterwards gets moved into the copy code (online change)
END_VAR
AddInput('ipContainer', ipContainer);
AddInput('hrPrev', hrPrev);
AddOutput('nNumberOfElements', nNumberOfElements);
AddOutput('hresult',hresult);
END_METHOD

METHOD PROTECTED OnExecute
hresult.Value := F_VN_GetNumberOfElements(
	ipContainer := ipContainer.Value,
    nNumberOfElements := nNumberOfElements.Value,
	hrPrev:= hrPrev.Value);
END_METHOD

METHOD PUBLIC PreExecutionCheck
VAR_INPUT
	Check : I_PreExecutionChecks;
END_VAR
Check.IsTrue(ipContainer.IsValid, 'ipContainer must be a valid container');
END_METHOD

END_FUNCTION_BLOCK

// ---- Nodes/Basic Container Ops/Node_F_VN_ExportSubContainer_String.TcPOU
{attribute 'linkalways'} 
{attribute 'no_explicit_call' := 'This FB is a CLASS and must be accessed using methods or properties'}
{attribute 'enable_dynamic_creation'}
FUNCTION_BLOCK Node_F_VN_ExportSubContainer_String EXTENDS VisionNode
VAR
    ipContainer : _ITcVnContainer;
    nIndex : _ULINT(0);
    sText : _STRING('');
    nMaxLength : _ULINT(0);
    hrPrev : _HRESULT(S_OK);
	hresult : _HRESULT(S_OK);
END_VAR

METHOD PUBLIC  Clone : I_Node
VAR
	pNode : POINTER TO Node_F_VN_ExportSubContainer_String;
END_VAR
pNode := __NEW(Node_F_VN_ExportSubContainer_String);
Clone := pNode^;
END_METHOD

METHOD FB_init : BOOL
VAR_INPUT
	bInitRetains : BOOL; // if TRUE, the retain variables are initialized (warm start / cold start)
	bInCopyCode : BOOL;  // if TRUE, the instance afterwards gets moved into the copy code (online change)
END_VAR
AddInput('ipContainer', ipContainer);
AddParameter('nIndex', nIndex);
AddParameter('nMaxLength', nMaxLength);
AddInput('hrPrev', hrPrev);
AddOutput('sText', sText);
AddOutput('hresult',hresult);
END_METHOD

METHOD PROTECTED OnExecute
hresult.Value := F_VN_ExportSubContainer_String(
	ipContainer := ipContainer.Value,
    nIndex := nIndex.Value,
    sText := sText.Value,
    nMaxLength := nMaxLength.Value,
	hrPrev:= hrPrev.Value);
END_METHOD

METHOD PUBLIC PreExecutionCheck
VAR_INPUT
	Check : I_PreExecutionChecks;
END_VAR
Check.IsTrue(ipContainer.IsValid, 'ipContainer must be a valid container');
Check.IsTrue(ipContainer.IsType(TC_GLOBAL_CONST_LIST.ContainerType_Vector_String_SINT), 'ipContainer contains incorrect type');
END_METHOD

END_FUNCTION_BLOCK

// ---- Nodes/Basic Container Ops/Node_F_VN_CheckIfEmpty.TcPOU
{attribute 'linkalways'} 
{attribute 'no_explicit_call' := 'This FB is a CLASS and must be accessed using methods or properties'}
{attribute 'enable_dynamic_creation'}
FUNCTION_BLOCK Node_F_VN_CheckIfEmpty EXTENDS VisionNode
VAR
    ipContainer : _ITcVnContainer;
    hrPrev : _HRESULT(S_OK);
	hresult : _HRESULT(S_OK);
END_VAR

METHOD PUBLIC  Clone : I_Node
VAR
	pNode : POINTER TO Node_F_VN_CheckIfEmpty;
END_VAR
pNode := __NEW(Node_F_VN_CheckIfEmpty);
Clone := pNode^;
END_METHOD

METHOD FB_init : BOOL
VAR_INPUT
	bInitRetains : BOOL; // if TRUE, the retain variables are initialized (warm start / cold start)
	bInCopyCode : BOOL;  // if TRUE, the instance afterwards gets moved into the copy code (online change)
END_VAR
AddInput('ipContainer', ipContainer);
AddInput('hrPrev', hrPrev);
AddOutput('hresult',hresult);
END_METHOD

METHOD PROTECTED OnExecute
hresult.Value := F_VN_CheckIfEmpty(
	ipContainer := ipContainer.Value,
	hrPrev:= hrPrev.Value);
END_METHOD

METHOD PUBLIC PreExecutionCheck
VAR_INPUT
	Check : I_PreExecutionChecks;
END_VAR
Check.IsTrue(ipContainer.IsValid, 'ipContainer must be a valid container');
END_METHOD

END_FUNCTION_BLOCK

// ---- Nodes/Basic Container Ops/Node_F_VN_CopyContainer.TcPOU
{attribute 'linkalways'} 
{attribute 'no_explicit_call' := 'This FB is a CLASS and must be accessed using methods or properties'}
{attribute 'enable_dynamic_creation'}
FUNCTION_BLOCK Node_F_VN_CopyContainer EXTENDS VisionNode
VAR
    ipSrcContainer : _ITcVnContainer;
    ipDestContainer : _ITcVnContainer;
    hrPrev : _HRESULT(S_OK);
	hresult : _HRESULT(S_OK);
END_VAR

METHOD PUBLIC  Clone : I_Node
VAR
	pNode : POINTER TO Node_F_VN_CopyContainer;
END_VAR
pNode := __NEW(Node_F_VN_CopyContainer);
Clone := pNode^;
END_METHOD

METHOD FB_init : BOOL
VAR_INPUT
	bInitRetains : BOOL; // if TRUE, the retain variables are initialized (warm start / cold start)
	bInCopyCode : BOOL;  // if TRUE, the instance afterwards gets moved into the copy code (online change)
END_VAR
AddInput('ipSrcContainer', ipSrcContainer);
AddInput('hrPrev', hrPrev);
AddOutput('ipDestContainer', ipDestContainer);
AddOutput('hresult',hresult);
END_METHOD

METHOD PROTECTED OnExecute
hresult.Value := F_VN_CopyContainer(
	ipSrcContainer := ipSrcContainer.Value,
    ipDestContainer := ipDestContainer.Value,
	hrPrev:= hrPrev.Value);
END_METHOD

METHOD PUBLIC PreExecutionCheck
VAR_INPUT
	Check : I_PreExecutionChecks;
END_VAR
Check.IsTrue(ipSrcContainer.IsValid, 'ipSrcContainer must be a valid container');
END_METHOD

END_FUNCTION_BLOCK

// ---- Nodes/Basic Image Ops/Node_F_VN_CreateNDimensionalImage.TcPOU
{attribute 'linkalways'} 
{attribute 'no_explicit_call' := 'This FB is a CLASS and must be accessed using methods or properties'}
{attribute 'enable_dynamic_creation'}
FUNCTION_BLOCK Node_F_VN_CreateNDimensionalImage EXTENDS VisionNode
VAR
    ipImage : _ITcVnImage;
    aShape : _TcVnArray33_UDINT;
    ePixelType : _ETcVnElementType(ETcVnElementType.TCVN_ET_USINT);
    hrPrev : _HRESULT(S_OK);
	hresult : _HRESULT(S_OK);
END_VAR

METHOD PUBLIC  Clone : I_Node
VAR
	pNode : POINTER TO Node_F_VN_CreateNDimensionalImage;
END_VAR
pNode := __NEW(Node_F_VN_CreateNDimensionalImage);
Clone := pNode^;
END_METHOD

METHOD FB_init : BOOL
VAR_INPUT
	bInitRetains : BOOL; // if TRUE, the retain variables are initialized (warm start / cold start)
	bInCopyCode : BOOL;  // if TRUE, the instance afterwards gets moved into the copy code (online change)
END_VAR
AddParameter('aShape', aShape);
AddParameter('ePixelType', ePixelType);
AddInput('hrPrev', hrPrev);
AddOutput('ipImage', ipImage);
AddOutput('hresult',hresult);
END_METHOD

METHOD PROTECTED OnExecute
hresult.Value := F_VN_CreateNDimensionalImage(
    ipImage := ipImage.Value,
    aShape := aShape.Value,
    ePixelType := ePixelType.Value,
	hrPrev:= hrPrev.Value);
END_METHOD

METHOD PUBLIC PreExecutionCheck
VAR_INPUT
	Check : I_PreExecutionChecks;
END_VAR
END_METHOD

END_FUNCTION_BLOCK

// ---- Nodes/Basic Image Ops/Node_F_VN_CreateNDimensionalImageAndSetPixels.TcPOU
{attribute 'linkalways'} 
{attribute 'no_explicit_call' := 'This FB is a CLASS and must be accessed using methods or properties'}
{attribute 'enable_dynamic_creation'}
FUNCTION_BLOCK Node_F_VN_CreateNDimensionalImageAndSetPixels EXTENDS VisionNode
VAR
    ipImage : _ITcVnImage;
    aShape : _TcVnArray33_UDINT;
    ePixelType : _ETcVnElementType(ETcVnElementType.TCVN_ET_USINT);
    fValue : _LREAL(0.0);
    hrPrev : _HRESULT(S_OK);
	hresult : _HRESULT(S_OK);
END_VAR

METHOD PUBLIC  Clone : I_Node
VAR
	pNode : POINTER TO Node_F_VN_CreateNDimensionalImageAndSetPixels;
END_VAR
pNode := __NEW(Node_F_VN_CreateNDimensionalImageAndSetPixels);
Clone := pNode^;
END_METHOD

METHOD FB_init : BOOL
VAR_INPUT
	bInitRetains : BOOL; // if TRUE, the retain variables are initialized (warm start / cold start)
	bInCopyCode : BOOL;  // if TRUE, the instance afterwards gets moved into the copy code (online change)
END_VAR
AddParameter('aShape', aShape);
AddParameter('ePixelType', ePixelType);
AddParameter('fValue', fValue);
AddInput('hrPrev', hrPrev);
AddOutput('ipImage', ipImage);
AddOutput('hresult',hresult);
END_METHOD

METHOD PROTECTED OnExecute
hresult.Value := F_VN_CreateNDimensionalImageAndSetPixels(
    ipImage := ipImage.Value,
    aShape := aShape.Value,
    ePixelType := ePixelType.Value,
    fValue := fValue.Value,
	hrPrev:= hrPrev.Value);
END_METHOD

METHOD PUBLIC PreExecutionCheck
VAR_INPUT
	Check : I_PreExecutionChecks;
END_VAR
END_METHOD

END_FUNCTION_BLOCK

// ---- Nodes/Basic Image Ops/Node_F_VN_ExportImageAsBmpSizeExp.TcPOU
{attribute 'linkalways'} 
{attribute 'no_explicit_call' := 'This FB is a CLASS and must be accessed using methods or properties'}
{attribute 'enable_dynamic_creation'}
FUNCTION_BLOCK Node_F_VN_ExportImageAsBmpSizeExp EXTENDS VisionNode
VAR
    ipImage : _ITcVnImage;
    nBufferSize : _ULINT(0);
    nWidth : _UDINT(0);
    nHeight : _UDINT(0);
    hrPrev : _HRESULT(S_OK);
	hresult : _HRESULT(S_OK);
END_VAR

METHOD PUBLIC  Clone : I_Node
VAR
	pNode : POINTER TO Node_F_VN_ExportImageAsBmpSizeExp;
END_VAR
pNode := __NEW(Node_F_VN_ExportImageAsBmpSizeExp);
Clone := pNode^;
END_METHOD

METHOD FB_init : BOOL
VAR_INPUT
	bInitRetains : BOOL; // if TRUE, the retain variables are initialized (warm start / cold start)
	bInCopyCode : BOOL;  // if TRUE, the instance afterwards gets moved into the copy code (online change)
END_VAR
AddInput('ipImage', ipImage);
AddParameter('nWidth', nWidth);
AddParameter('nHeight', nHeight);
AddInput('hrPrev', hrPrev);
AddOutput('nBufferSize', nBufferSize);
AddOutput('hresult', hresult);
END_METHOD

METHOD PROTECTED OnExecute
hresult.Value := F_VN_ExportImageAsBmpSizeExp(
    ipImage := ipImage.Value,
    nBufferSize := nBufferSize.Value,
    nWidth := nWidth.Value,
    nHeight := nHeight.Value,
	hrPrev:= hrPrev.Value);
END_METHOD

METHOD PUBLIC PreExecutionCheck
VAR_INPUT
	Check : I_PreExecutionChecks;
END_VAR
Check.IsTrue(ipImage.IsValid, 'ipImage must contain an image');
END_METHOD

END_FUNCTION_BLOCK

// ---- Nodes/Basic Image Ops/Node_F_VN_FuseImages.TcPOU
{attribute 'linkalways'} 
{attribute 'no_explicit_call' := 'This FB is a CLASS and must be accessed using methods or properties'}
{attribute 'enable_dynamic_creation'}
FUNCTION_BLOCK Node_F_VN_FuseImages EXTENDS VisionNode
VAR
    ipSrcImage1 : _ITcVnImage;
    ipSrcImage2 : _ITcVnImage;
    ipDestImage : _ITcVnImage;
    nFirstLine : _UDINT(0);
    nNumLines : _UDINT(0);
    hrPrev : _HRESULT(S_OK);
	hresult : _HRESULT(S_OK);
END_VAR

METHOD PUBLIC  Clone : I_Node
VAR
	pNode : POINTER TO Node_F_VN_FuseImages;
END_VAR
pNode := __NEW(Node_F_VN_FuseImages);
Clone := pNode^;
END_METHOD

METHOD FB_init : BOOL
VAR_INPUT
	bInitRetains : BOOL; // if TRUE, the retain variables are initialized (warm start / cold start)
	bInCopyCode : BOOL;  // if TRUE, the instance afterwards gets moved into the copy code (online change)
END_VAR
AddInput('ipSrcImage1', ipSrcImage1);
AddInput('ipSrcImage2', ipSrcImage2);
AddParameter('nFirstLine', nFirstLine);
AddParameter('nNumLines', nNumLines);
AddInput('hrPrev', hrPrev);
AddOutput('ipDestImage', ipDestImage);
AddOutput('hresult',hresult);
END_METHOD

METHOD PROTECTED OnExecute
hresult.Value := F_VN_FuseImages(
    ipSrcImage1 := ipSrcImage1.Value,
    ipSrcImage2 := ipSrcImage2.Value,
	ipDestImage := ipDestImage.Value,
    nFirstLine := nFirstLine.Value,
    nNumLines := nNumLines.Value,
	hrPrev:= hrPrev.Value);
END_METHOD

METHOD PUBLIC PreExecutionCheck
VAR_INPUT
	Check : I_PreExecutionChecks;
END_VAR
Check.IsTrue(ipSrcImage1.IsValid, 'ipSrcImage1 must contain an image');
Check.IsTrue(ipSrcImage2.IsValid, 'ipSrcImage2 must contain an image');
Check.IsTrue(IsImage1WidthEqualToImage2Width(ipSrcImage1.Value, ipSrcImage2.Value), 'ipSrcImage1 must be the same width as ipSrcImage2');
Check.IsTrue(ImagesHaveMatchingPixelFormats(ipSrcImage1.Value, ipSrcImage2.Value), 'ipSrcImage2 must have same pixel depth as ipSrcImage1');
END_METHOD

END_FUNCTION_BLOCK

// ---- Nodes/Basic Image Ops/Node_F_VN_CopyImageRegion.TcPOU
{attribute 'linkalways'} 
{attribute 'no_explicit_call' := 'This FB is a CLASS and must be accessed using methods or properties'}
{attribute 'enable_dynamic_creation'}
FUNCTION_BLOCK Node_F_VN_CopyImageRegion EXTENDS VisionNode
VAR
    ipSrcImage : _ITcVnImage;
    nX : _UDINT(0);
    nY : _UDINT(0);
    nWidth : _UDINT(0);
    nHeight : _UDINT(0);
    ipDestImage : _ITcVnImage;
    hrPrev : _HRESULT(S_OK);
	hresult : _HRESULT(S_OK);
END_VAR

METHOD PUBLIC  Clone : I_Node
VAR
	pNode : POINTER TO Node_F_VN_CopyImageRegion;
END_VAR
pNode := __NEW(Node_F_VN_CopyImageRegion);
Clone := pNode^;
END_METHOD

METHOD FB_init : BOOL
VAR_INPUT
	bInitRetains : BOOL; // if TRUE, the retain variables are initialized (warm start / cold start)
	bInCopyCode : BOOL;  // if TRUE, the instance afterwards gets moved into the copy code (online change)
END_VAR
AddInput('ipSrcImage', ipSrcImage);
AddParameter('nX', nX);
AddParameter('nY', nY);
AddParameter('nWidth', nWidth);
AddParameter('nHeight', nHeight);
AddInput('hrPrev', hrPrev);
AddOutput('ipDestImage', ipDestImage);
AddOutput('hresult',hresult);
END_METHOD

METHOD PROTECTED OnExecute
hresult.Value := F_VN_CopyImageRegion(
    ipSrcImage := ipSrcImage.Value,
    nX := nX.Value,
    nY := nY.Value,
    nWidth := nWidth.Value,
	nHeight := nHeight.Value,
	ipDestImage := ipDestImage.Value,
	hrPrev:= hrPrev.Value);
END_METHOD

METHOD PUBLIC PreExecutionCheck
VAR_INPUT
	Check : I_PreExecutionChecks;
END_VAR
VAR
    imageWidth : UDINT;
    imageHeight : UDINT;
    roiRectangle : TcVnRectangle_UDINT;
END_VAR
Check.IsTrue(ipSrcImage.IsValid, 'ipSrcImage must contain an image');

IF Check.Failed THEN
    RETURN;
END_IF

ipSrcImage.Value.GetWidth(imageWidth);
ipSrcImage.Value.GetHeight(imageHeight);
roiRectangle.nX := nX.Value;
roiRectangle.nY := nY.Value;
roiRectangle.nWidth := nWidth.Value;
roiRectangle.nHeight := nHeight.Value;

Check.IsTrue((roiRectangle.nWidth <= imageWidth), 'ROI width must not be greater than image width');
Check.IsTrue((roiRectangle.nWidth <= (imageWidth - roiRectangle.nX)), 'ROI too wide to fit within image');
Check.IsTrue((roiRectangle.nHeight <= imageHeight), 'ROI height must not be greater than image height');
Check.IsTrue((roiRectangle.nHeight <= (imageHeight - roiRectangle.nY)), 'ROI too high to fit within image');
END_METHOD

END_FUNCTION_BLOCK

// ---- Nodes/Basic Image Ops/Node_F_VN_CopyImageRegionToRegion.TcPOU
{attribute 'linkalways'} 
{attribute 'no_explicit_call' := 'This FB is a CLASS and must be accessed using methods or properties'}
{attribute 'enable_dynamic_creation'}
FUNCTION_BLOCK Node_F_VN_CopyImageRegionToRegion EXTENDS VisionNode
VAR
    ipSrcImage : _ITcVnImage;
    nXSrc : _UDINT(0);
    nYSrc : _UDINT(0);
    nWidth : _UDINT(0);
    nHeight : _UDINT(0);
    ipDestImage : _ITcVnImage;
    nXDest : _UDINT(0);
    nYDest : _UDINT(0);
    hrPrev : _HRESULT(S_OK);
	hresult : _HRESULT(S_OK);
END_VAR

METHOD PUBLIC  Clone : I_Node
VAR
	pNode : POINTER TO Node_F_VN_CopyImageRegionToRegion;
END_VAR
pNode := __NEW(Node_F_VN_CopyImageRegionToRegion);
Clone := pNode^;
END_METHOD

METHOD FB_init : BOOL
VAR_INPUT
	bInitRetains : BOOL; // if TRUE, the retain variables are initialized (warm start / cold start)
	bInCopyCode : BOOL;  // if TRUE, the instance afterwards gets moved into the copy code (online change)
END_VAR
AddInput('ipSrcImage', ipSrcImage);
AddParameter('nXSrc', nXSrc);
AddParameter('nYSrc', nYSrc);
AddParameter('nWidth', nWidth);
AddParameter('nHeight', nHeight);
AddInput('ipDestImage', ipDestImage);
AddParameter('nXDest', nXDest);
AddParameter('nYDest', nYDest);
AddInput('hrPrev', hrPrev);
AddOutput('ipDestImage', ipDestImage);
AddOutput('hresult',hresult);
END_METHOD

METHOD PROTECTED OnExecute
hresult.Value := F_VN_CopyImageRegionToRegion(
    ipSrcImage := ipSrcImage.Value,
    nXSrc := nXSrc.Value,
    nYSrc := nYSrc.Value,
    nWidth := nWidth.Value,
	nHeight := nHeight.Value,
	ipDestImage := ipDestImage.Value,
    nXDest := nXDest.Value,
    nYDest := nYDest.Value,
	hrPrev:= hrPrev.Value);
END_METHOD

METHOD PUBLIC PreExecutionCheck
VAR_INPUT
	Check : I_PreExecutionChecks;
END_VAR
VAR
    imgWidth : UDINT;
    imgHeight : UDINT;
    roiRectangle : TcVnRectangle_UDINT;
END_VAR
Check.IsTrue(ipSrcImage.IsValid, 'ipSrcImage must contain an image');

IF Check.Failed THEN
    RETURN;
END_IF

ipSrcImage.Value.GetWidth(imgWidth);
ipSrcImage.Value.GetHeight(imgHeight);
roiRectangle.nX := nXSrc.Value;
roiRectangle.nY := nYSrc.Value;
roiRectangle.nWidth := nWidth.Value;
roiRectangle.nHeight := nHeight.Value;

Check.IsTrue(IsRoiSizeOK_Udint(roiRectangle, imgWidth, imgHeight), 'ROI must fit within ipSrcImage');

//TODO Check nXDist and nYDest values?
END_METHOD

END_FUNCTION_BLOCK

// ---- Nodes/Basic Image Ops/Node_F_VN_ExportImageSize.TcPOU
{attribute 'linkalways'} 
{attribute 'no_explicit_call' := 'This FB is a CLASS and must be accessed using methods or properties'}
{attribute 'enable_dynamic_creation'}
FUNCTION_BLOCK Node_F_VN_ExportImageSize EXTENDS VisionNode
VAR
    ipImage : _ITcVnImage;
    nBufferSize : _ULINT(0);
    hrPrev : _HRESULT(S_OK);
	hresult : _HRESULT(S_OK);
END_VAR

METHOD PUBLIC  Clone : I_Node
VAR
	pNode : POINTER TO Node_F_VN_ExportImageSize;
END_VAR
pNode := __NEW(Node_F_VN_ExportImageSize);
Clone := pNode^;
END_METHOD

METHOD FB_init : BOOL
VAR_INPUT
	bInitRetains : BOOL; // if TRUE, the retain variables are initialized (warm start / cold start)
	bInCopyCode : BOOL;  // if TRUE, the instance afterwards gets moved into the copy code (online change)
END_VAR
AddInput('ipImage', ipImage);
AddInput('hrPrev', hrPrev);
AddOutput('nBufferSize', nBufferSize);
AddOutput('hresult',hresult);
END_METHOD

METHOD PROTECTED OnExecute
hresult.Value := F_VN_ExportImageSize(
    ipImage := ipImage.Value,
    nBufferSize := nBufferSize.Value,
	hrPrev:= hrPrev.Value);
END_METHOD

METHOD PUBLIC PreExecutionCheck
VAR_INPUT
	Check : I_PreExecutionChecks;
END_VAR
Check.IsTrue(ipImage.IsValid, 'ipImage must contain an image');
END_METHOD

END_FUNCTION_BLOCK

// ---- Nodes/Basic Image Ops/Node_F_VN_ExportImageAsBmpSize.TcPOU
{attribute 'linkalways'} 
{attribute 'no_explicit_call' := 'This FB is a CLASS and must be accessed using methods or properties'}
{attribute 'enable_dynamic_creation'}
FUNCTION_BLOCK Node_F_VN_ExportImageAsBmpSize EXTENDS VisionNode
VAR
    ipImage : _ITcVnImage;
    nBufferSize : _ULINT(0);
    hrPrev : _HRESULT(S_OK);
	hresult : _HRESULT(S_OK);
END_VAR

METHOD PUBLIC  Clone : I_Node
VAR
	pNode : POINTER TO Node_F_VN_ExportImageAsBmpSize;
END_VAR
pNode := __NEW(Node_F_VN_ExportImageAsBmpSize);
Clone := pNode^;
END_METHOD

METHOD FB_init : BOOL
VAR_INPUT
	bInitRetains : BOOL; // if TRUE, the retain variables are initialized (warm start / cold start)
	bInCopyCode : BOOL;  // if TRUE, the instance afterwards gets moved into the copy code (online change)
END_VAR
AddInput('ipImage', ipImage);
AddInput('hrPrev', hrPrev);
AddOutput('nBufferSize', nBufferSize);
AddOutput('hresult',hresult);
END_METHOD

METHOD PROTECTED OnExecute
hresult.Value := F_VN_ExportImageAsBmpSize(
    ipImage := ipImage.Value,
    nBufferSize := nBufferSize.Value,
	hrPrev:= hrPrev.Value);
END_METHOD

METHOD PUBLIC PreExecutionCheck
VAR_INPUT
	Check : I_PreExecutionChecks;
END_VAR
Check.IsTrue(ipImage.IsValid, 'ipImage must contain an image');
END_METHOD

END_FUNCTION_BLOCK

// ---- Nodes/Basic Image Ops/Node_F_VN_MixImageChannels.TcPOU
{attribute 'linkalways'} 
{attribute 'no_explicit_call' := 'This FB is a CLASS and must be accessed using methods or properties'}
{attribute 'enable_dynamic_creation'}
FUNCTION_BLOCK Node_F_VN_MixImageChannels EXTENDS VisionNode
VAR
    ipSrcImage : _ITcVnImage;
    ipDestImage : _ITcVnImage;
    ipIndicesFromTo : _ITcVnContainer;
    hrPrev : _HRESULT(S_OK);
	hresult : _HRESULT(S_OK);
END_VAR

METHOD PUBLIC  Clone : I_Node
VAR
	pNode : POINTER TO Node_F_VN_MixImageChannels;
END_VAR
pNode := __NEW(Node_F_VN_MixImageChannels);
Clone := pNode^;
END_METHOD

METHOD FB_init : BOOL
VAR_INPUT
	bInitRetains : BOOL; // if TRUE, the retain variables are initialized (warm start / cold start)
	bInCopyCode : BOOL;  // if TRUE, the instance afterwards gets moved into the copy code (online change)
END_VAR
AddInput('ipSrcImage', ipSrcImage);
AddInput('ipIndicesFromTo', ipIndicesFromTo);
AddInput('hrPrev', hrPrev);
AddOutput('ipDestImage', ipDestImage);
AddOutput('hresult',hresult);
END_METHOD

METHOD PROTECTED OnExecute
hresult.Value := F_VN_MixImageChannels(
    ipSrcImage := ipSrcImage.Value,
	ipDestImage := ipDestImage.Value,
    ipIndicesFromTo := ipIndicesFromTo.Value,
	hrPrev := hrPrev.Value);
END_METHOD

METHOD PUBLIC PreExecutionCheck
VAR_INPUT
	Check : I_PreExecutionChecks;
END_VAR
Check.IsTrue(ipSrcImage.IsValid, 'ipSrcImage must contain an image');
Check.IsTrue(ipIndicesFromTo.IsType(TC_GLOBAL_CONST_LIST.ContainerType_Vector_TcVnVector2_DINT),
              'ipIndicesFromTo contains incorrect type');
END_METHOD

END_FUNCTION_BLOCK

// ---- Nodes/Basic Image Ops/Node_F_VN_GetLayoutInfo.TcPOU
{attribute 'linkalways'} 
{attribute 'no_explicit_call' := 'This FB is a CLASS and must be accessed using methods or properties'}
{attribute 'enable_dynamic_creation'}
FUNCTION_BLOCK Node_F_VN_GetLayoutInfo EXTENDS VisionNode
VAR
    ipImage : _ITcVnImage;
    aLayoutInfo : _TcVnArray33_UDINT;
    hrPrev : _HRESULT(S_OK);
	hresult : _HRESULT(S_OK);
END_VAR

METHOD PUBLIC  Clone : I_Node
VAR
	pNode : POINTER TO Node_F_VN_GetLayoutInfo;
END_VAR
pNode := __NEW(Node_F_VN_GetLayoutInfo);
Clone := pNode^;
END_METHOD

METHOD FB_init : BOOL
VAR_INPUT
	bInitRetains : BOOL; // if TRUE, the retain variables are initialized (warm start / cold start)
	bInCopyCode : BOOL;  // if TRUE, the instance afterwards gets moved into the copy code (online change)
END_VAR
AddInput('ipImage', ipImage);
AddInput('hrPrev', hrPrev);
AddOutput('aLayoutInfo', aLayoutInfo);
AddOutput('hresult',hresult);
END_METHOD

METHOD PROTECTED OnExecute
hresult.Value := F_VN_GetLayoutInfo(
    ipImage := ipImage.Value,
	aLayoutInfo := aLayoutInfo.Value,
	hrPrev:= hrPrev.Value);
END_METHOD

METHOD PUBLIC PreExecutionCheck
VAR_INPUT
	Check : I_PreExecutionChecks;
END_VAR
Check.IsTrue(ipImage.IsValid, 'ipImage must contain an image');
END_METHOD

END_FUNCTION_BLOCK

// ---- Nodes/Basic Image Ops/Node_F_VN_PadImageBorder.TcPOU
{attribute 'linkalways'} 
{attribute 'no_explicit_call' := 'This FB is a CLASS and must be accessed using methods or properties'}
{attribute 'enable_dynamic_creation'}
FUNCTION_BLOCK Node_F_VN_PadImageBorder EXTENDS VisionNode
VAR
    ipSrcImage : _ITcVnImage;
    ipPaddedImage : _ITcVnImage;
    nTopBorder : _UDINT(0);
    nBottomBorder : _UDINT(0);
    nLeftBorder : _UDINT(0);
    nRightBorder : _UDINT(0);
    hrPrev : _HRESULT(S_OK);
	hresult : _HRESULT(S_OK);
END_VAR

METHOD PUBLIC  Clone : I_Node
VAR
	pNode : POINTER TO Node_F_VN_PadImageBorder;
END_VAR
pNode := __NEW(Node_F_VN_PadImageBorder);
Clone := pNode^;
END_METHOD

METHOD FB_init : BOOL
VAR_INPUT
	bInitRetains : BOOL; // if TRUE, the retain variables are initialized (warm start / cold start)
	bInCopyCode : BOOL;  // if TRUE, the instance afterwards gets moved into the copy code (online change)
END_VAR
AddInput('ipSrcImage', ipSrcImage);
AddParameter('nTopBorder', nTopBorder);
AddParameter('nBottomBorder', nBottomBorder);
AddParameter('nLeftBorder', nLeftBorder);
AddParameter('nRightBorder', nRightBorder);
AddInput('hrPrev', hrPrev);
AddOutput('ipPaddedImage', ipPaddedImage);
AddOutput('hresult',hresult);
END_METHOD

METHOD PROTECTED OnExecute
hresult.Value := F_VN_PadImageBorder(
    ipSrcImage := ipSrcImage.Value,
	ipPaddedImage := ipPaddedImage.Value,
    nTopBorder := nTopBorder.Value,
    nBottomBorder := nBottomBorder.Value,
    nLeftBorder := nLeftBorder.Value,
    nRightBorder := nRightBorder.Value,
	hrPrev:= hrPrev.Value);
END_METHOD

METHOD PUBLIC PreExecutionCheck
VAR_INPUT
	Check : I_PreExecutionChecks;
END_VAR
Check.IsTrue(ipSrcImage.IsValid, 'ipSrcImage must contain an image');
END_METHOD

END_FUNCTION_BLOCK

// ---- Nodes/Basic Image Ops/Node_F_VN_PadImageBorderExp.TcPOU
{attribute 'linkalways'} 
{attribute 'no_explicit_call' := 'This FB is a CLASS and must be accessed using methods or properties'}
{attribute 'enable_dynamic_creation'}
FUNCTION_BLOCK Node_F_VN_PadImageBorderExp EXTENDS VisionNode
VAR
    ipSrcImage : _ITcVnImage;
    ipPaddedImage : _ITcVnImage;
    nTopBorder : _UDINT(0);
    nBottomBorder : _UDINT(0);
    nLeftBorder : _UDINT(0);
    nRightBorder : _UDINT(0);
    ePaddingType : _ETcVnBorderInterpolationMethod(ETcVnBorderInterpolationMethod.TCVN_BIM_CONSTANT);
    aPaddingValue : _TcVnVector4_LREAL;
    hrPrev : _HRESULT(S_OK);
	hresult : _HRESULT(S_OK);
END_VAR

METHOD PUBLIC  Clone : I_Node
VAR
	pNode : POINTER TO Node_F_VN_PadImageBorderExp;
END_VAR
pNode := __NEW(Node_F_VN_PadImageBorderExp);
Clone := pNode^;
END_METHOD

METHOD FB_init : BOOL
VAR_INPUT
	bInitRetains : BOOL; // if TRUE, the retain variables are initialized (warm start / cold start)
	bInCopyCode : BOOL;  // if TRUE, the instance afterwards gets moved into the copy code (online change)
END_VAR
AddInput('ipSrcImage', ipSrcImage);
AddParameter('nTopBorder', nTopBorder);
AddParameter('nBottomBorder', nBottomBorder);
AddParameter('nLeftBorder', nLeftBorder);
AddParameter('nRightBorder', nRightBorder);
AddParameter('ePaddingType', ePaddingType);
AddInput('aPaddingValue', aPaddingValue);
AddInput('hrPrev', hrPrev);
AddOutput('ipPaddedImage', ipPaddedImage);
AddOutput('hresult',hresult);
END_METHOD

METHOD PROTECTED OnExecute
hresult.Value := F_VN_PadImageBorderExp(
    ipSrcImage := ipSrcImage.Value,
	ipPaddedImage := ipPaddedImage.Value,
    nTopBorder := nTopBorder.Value,
    nBottomBorder := nBottomBorder.Value,
    nLeftBorder := nLeftBorder.Value,
    nRightBorder := nRightBorder.Value,
    ePaddingType := ePaddingType.Value,
    aPaddingValue := aPaddingValue.Value,
	hrPrev:= hrPrev.Value);
END_METHOD

METHOD PUBLIC PreExecutionCheck
VAR_INPUT
	Check : I_PreExecutionChecks;
END_VAR
Check.IsTrue(ipSrcImage.IsValid, 'ipSrcImage must contain an image');
END_METHOD

END_FUNCTION_BLOCK

// ---- Nodes/Basic Image Ops/Node_F_VN_SetImageChannel.TcPOU
{attribute 'linkalways'} 
{attribute 'no_explicit_call' := 'This FB is a CLASS and must be accessed using methods or properties'}
{attribute 'enable_dynamic_creation'}
FUNCTION_BLOCK Node_F_VN_SetImageChannel EXTENDS VisionNode
VAR
    ipSrcImage : _ITcVnImage;
    ipDestImage : _ITcVnImage;
    nSrcChannelIndex : _UINT(0);
    nDestChannelIndex : _UINT(0);
    hrPrev : _HRESULT(S_OK);
	hresult : _HRESULT(S_OK);
END_VAR

METHOD PUBLIC  Clone : I_Node
VAR
	pNode : POINTER TO Node_F_VN_SetImageChannel;
END_VAR
pNode := __NEW(Node_F_VN_SetImageChannel);
Clone := pNode^;
END_METHOD

METHOD FB_init : BOOL
VAR_INPUT
	bInitRetains : BOOL; // if TRUE, the retain variables are initialized (warm start / cold start)
	bInCopyCode : BOOL;  // if TRUE, the instance afterwards gets moved into the copy code (online change)
END_VAR
AddInput('ipSrcImage', ipSrcImage);
AddInput('ipDestImage', ipDestImage);
AddParameter('nSrcChannelIndex', nSrcChannelIndex);
AddParameter('nDestChannelIndex', nDestChannelIndex);
AddInput('hrPrev', hrPrev);
AddOutput('ipDestImage', ipDestImage);
AddOutput('hresult',hresult);
END_METHOD

METHOD PROTECTED OnExecute
hresult.Value := F_VN_SetImageChannel(
    ipSrcImage := ipSrcImage.Value,
	ipDestImage := ipDestImage.Value,
    nSrcChannelIndex := nSrcChannelIndex.Value,
    nDestChannelIndex := nDestChannelIndex.Value,
	hrPrev:= hrPrev.Value);
END_METHOD

METHOD PUBLIC PreExecutionCheck
VAR_INPUT
	Check : I_PreExecutionChecks;
END_VAR
VAR
	srcImageInfo : TcVnImageInfo;
	destImageInfo : TcVnImageInfo;
END_VAR
Check.IsTrue(ipSrcImage.IsValid, 'ipSrcImage must contain an image');

IF ipSrcImage.TryGetImageInfo(srcImageInfo) THEN
	Check.IsTrue((nSrcChannelIndex.Value <= srcImageInfo.stPixelFormat.nChannels), 'nSrcChannelIndex is greater than the available ipSrcImage channels');
END_IF

IF NOT ipDestImage.IsValid THEN
	RETURN;
END_IF

IF ipDestImage.TryGetImageInfo(destImageInfo) THEN
	Check.IsTrue((nDestChannelIndex.Value <= destImageInfo.stPixelFormat.nChannels), 'nDestChannelIndex is greater than the available ipDestImage channels');
END_IF

